FONT_16X26:ARRAY[0..255,0..51]OF BYTE :=[
16#00,16#00,16#00,16#00,16#00,16#00,16#00,16#00,16#00,16#00,16#00,16#00,16#00,16#00,16#00,16#00,16#00,16#00,16#00,16#00,16#00,16#00,16#00,16#00,16#00,16#00,16#00,16#00,16#00,16#00,16#00,16#00,16#00,16#00,16#00,16#00,16#00,16#00,16#00,16#00,16#00,16#00,16#00,16#00,16#00,16#00,16#00,16#00,16#00,16#00,16#00,16#00,	// 16#00
16#00,16#00,16#00,16#00,16#00,16#00,16#00,16#00,16#00,16#00,16#00,16#00,16#00,16#00,16#E0,16#07,16#30,16#0C,16#08,16#10,16#64,16#26,16#66,16#66,16#02,16#40,16#02,16#40,16#12,16#48,16#12,16#48,16#36,16#6C,16#24,16#24,16#C8,16#13,16#30,16#0C,16#E0,16#07,16#00,16#00,16#00,16#00,16#00,16#00,16#00,16#00,16#00,16#00,	// 16#01
16#00,16#00,16#00,16#00,16#00,16#00,16#00,16#00,16#00,16#00,16#00,16#00,16#00,16#00,16#E0,16#07,16#F0,16#0F,16#F8,16#1F,16#FC,16#3F,16#9E,16#79,16#9E,16#79,16#FE,16#7F,16#FE,16#7F,16#EE,16#77,16#EE,16#77,16#DC,16#3B,16#38,16#1C,16#F0,16#0F,16#E0,16#07,16#00,16#00,16#00,16#00,16#00,16#00,16#00,16#00,16#00,16#00,	// 16#02
16#00,16#00,16#00,16#00,16#3C,16#3C,16#7E,16#7E,16#FE,16#7F,16#FF,16#FF,16#FF,16#FF,16#FF,16#FF,16#FF,16#FF,16#FF,16#FF,16#FF,16#FF,16#FE,16#7F,16#FE,16#7F,16#FC,16#3F,16#FC,16#3F,16#F8,16#1F,16#F0,16#0F,16#F0,16#0F,16#E0,16#07,16#C0,16#03,16#80,16#01,16#00,16#00,16#00,16#00,16#00,16#00,16#00,16#00,16#00,16#00,	// 16#03
16#00,16#00,16#00,16#00,16#00,16#01,16#80,16#01,16#80,16#03,16#C0,16#07,16#E0,16#07,16#F0,16#0F,16#F8,16#1F,16#FC,16#3F,16#FE,16#7F,16#FF,16#FF,16#FE,16#7F,16#FC,16#3F,16#F8,16#1F,16#F0,16#0F,16#E0,16#07,16#C0,16#07,16#80,16#03,16#80,16#01,16#00,16#01,16#00,16#00,16#00,16#00,16#00,16#00,16#00,16#00,16#00,16#00,	// 16#04
16#00,16#00,16#00,16#00,16#C0,16#03,16#E0,16#07,16#F0,16#0F,16#F0,16#0F,16#F0,16#0F,16#F0,16#0F,16#E0,16#07,16#FC,16#3F,16#FE,16#7F,16#FF,16#FF,16#FF,16#FF,16#FF,16#FF,16#FE,16#7F,16#9C,16#39,16#80,16#01,16#80,16#01,16#C0,16#03,16#C0,16#03,16#C0,16#03,16#00,16#00,16#00,16#00,16#00,16#00,16#00,16#00,16#00,16#00,	// 16#05
16#00,16#00,16#00,16#00,16#80,16#00,16#80,16#01,16#C0,16#01,16#E0,16#03,16#F0,16#07,16#F0,16#0F,16#F8,16#1F,16#FC,16#3F,16#FE,16#7F,16#FF,16#7F,16#FF,16#FF,16#FF,16#FF,16#FF,16#FF,16#FE,16#7F,16#9C,16#39,16#80,16#01,16#80,16#01,16#C0,16#03,16#C0,16#03,16#00,16#00,16#00,16#00,16#00,16#00,16#00,16#00,16#00,16#00,	// 16#06
16#00,16#00,16#00,16#00,16#00,16#00,16#00,16#00,16#00,16#00,16#00,16#00,16#00,16#00,16#00,16#00,16#00,16#00,16#00,16#00,16#00,16#00,16#00,16#00,16#00,16#00,16#00,16#00,16#00,16#00,16#00,16#00,16#00,16#00,16#00,16#00,16#00,16#00,16#00,16#00,16#00,16#00,16#00,16#00,16#00,16#00,16#00,16#00,16#00,16#00,16#00,16#00,	// 16#07
16#00,16#00,16#00,16#00,16#00,16#00,16#00,16#00,16#00,16#00,16#00,16#00,16#00,16#00,16#00,16#00,16#00,16#00,16#00,16#00,16#00,16#00,16#00,16#00,16#00,16#00,16#00,16#00,16#00,16#00,16#00,16#00,16#00,16#00,16#00,16#00,16#00,16#00,16#00,16#00,16#00,16#00,16#00,16#00,16#00,16#00,16#00,16#00,16#00,16#00,16#00,16#00,	// 16#08
16#00,16#00,16#00,16#00,16#00,16#00,16#00,16#00,16#00,16#00,16#00,16#00,16#00,16#00,16#00,16#00,16#00,16#00,16#00,16#00,16#00,16#00,16#00,16#00,16#00,16#00,16#00,16#00,16#00,16#00,16#00,16#00,16#00,16#00,16#00,16#00,16#00,16#00,16#00,16#00,16#00,16#00,16#00,16#00,16#00,16#00,16#00,16#00,16#00,16#00,16#00,16#00,	// 16#09
16#00,16#00,16#00,16#00,16#00,16#00,16#00,16#00,16#00,16#00,16#00,16#00,16#00,16#00,16#00,16#00,16#00,16#00,16#00,16#00,16#00,16#00,16#00,16#00,16#00,16#00,16#00,16#00,16#00,16#00,16#00,16#00,16#00,16#00,16#00,16#00,16#00,16#00,16#00,16#00,16#00,16#00,16#00,16#00,16#00,16#00,16#00,16#00,16#00,16#00,16#00,16#00,	// 16#0A
16#00,16#00,16#00,16#00,16#0C,16#00,16#FE,16#00,16#FE,16#00,16#1E,16#00,16#33,16#00,16#73,16#00,16#E0,16#0F,16#E0,16#3F,16#70,16#70,16#30,16#60,16#18,16#C0,16#18,16#C0,16#18,16#C0,16#18,16#C0,16#18,16#C0,16#30,16#60,16#70,16#70,16#E0,16#3F,16#80,16#0F,16#00,16#00,16#00,16#00,16#00,16#00,16#00,16#00,16#00,16#00,	// 16#0B
16#00,16#00,16#00,16#00,16#E0,16#03,16#F8,16#0F,16#1C,16#1C,16#0C,16#18,16#06,16#30,16#06,16#30,16#06,16#30,16#06,16#30,16#06,16#38,16#0C,16#18,16#1C,16#1E,16#F8,16#0F,16#F0,16#03,16#C0,16#00,16#C0,16#00,16#F8,16#07,16#F8,16#07,16#C0,16#00,16#C0,16#00,16#00,16#00,16#00,16#00,16#00,16#00,16#00,16#00,16#00,16#00,	// 16#0C
16#00,16#00,16#00,16#00,16#00,16#00,16#00,16#00,16#00,16#00,16#00,16#00,16#00,16#00,16#00,16#00,16#00,16#00,16#00,16#00,16#00,16#00,16#00,16#00,16#00,16#00,16#00,16#00,16#00,16#00,16#00,16#00,16#00,16#00,16#00,16#00,16#00,16#00,16#00,16#00,16#00,16#00,16#00,16#00,16#00,16#00,16#00,16#00,16#00,16#00,16#00,16#00,	// 16#0D
16#00,16#00,16#00,16#00,16#02,16#00,16#0E,16#00,16#7E,16#00,16#FE,16#01,16#E2,16#07,16#82,16#07,16#02,16#04,16#02,16#04,16#02,16#04,16#02,16#04,16#02,16#04,16#02,16#04,16#02,16#04,16#02,16#04,16#1E,16#04,16#3E,16#04,16#7E,16#04,16#7C,16#04,16#38,16#3C,16#00,16#7C,16#00,16#FC,16#00,16#F8,16#00,16#70,16#00,16#00,	// 16#0E
16#00,16#00,16#00,16#00,16#00,16#00,16#00,16#00,16#00,16#00,16#80,16#01,16#88,16#11,16#DC,16#3B,16#F8,16#1F,16#30,16#0C,16#18,16#18,16#1E,16#78,16#1E,16#78,16#18,16#18,16#30,16#0C,16#F8,16#1F,16#DC,16#3B,16#88,16#11,16#80,16#01,16#00,16#00,16#00,16#00,16#00,16#00,16#00,16#00,16#00,16#00,16#00,16#00,16#00,16#00,	// 16#0F
16#00,16#00,16#00,16#00,16#00,16#00,16#00,16#00,16#00,16#00,16#00,16#00,16#00,16#40,16#00,16#70,16#00,16#7C,16#00,16#7F,16#80,16#7F,16#E0,16#7F,16#F8,16#7F,16#FE,16#7F,16#F8,16#7F,16#E0,16#7F,16#80,16#7F,16#00,16#7F,16#00,16#7C,16#00,16#70,16#00,16#40,16#00,16#00,16#00,16#00,16#00,16#00,16#00,16#00,16#00,16#00,	// 16#10
16#00,16#00,16#00,16#00,16#00,16#00,16#00,16#00,16#00,16#00,16#00,16#00,16#02,16#00,16#0E,16#00,16#3E,16#00,16#FE,16#00,16#FE,16#01,16#FE,16#07,16#FE,16#1F,16#FE,16#7F,16#FE,16#1F,16#FE,16#07,16#FE,16#01,16#FE,16#00,16#3E,16#00,16#0E,16#00,16#02,16#00,16#00,16#00,16#00,16#00,16#00,16#00,16#00,16#00,16#00,16#00,	// 16#11
16#00,16#00,16#00,16#00,16#80,16#01,16#80,16#01,16#C0,16#03,16#E0,16#07,16#B0,16#0D,16#80,16#01,16#80,16#01,16#80,16#01,16#80,16#01,16#80,16#01,16#80,16#01,16#80,16#01,16#80,16#01,16#80,16#01,16#80,16#01,16#80,16#01,16#80,16#01,16#80,16#01,16#B0,16#0D,16#E0,16#07,16#C0,16#03,16#80,16#01,16#80,16#01,16#00,16#00,	// 16#12
16#00,16#00,16#00,16#00,16#38,16#0E,16#38,16#0E,16#38,16#0E,16#38,16#0E,16#38,16#0E,16#38,16#0E,16#38,16#0E,16#38,16#0E,16#38,16#0E,16#38,16#0E,16#38,16#0E,16#38,16#0E,16#38,16#0E,16#38,16#0E,16#00,16#00,16#00,16#00,16#38,16#0E,16#38,16#0E,16#38,16#0E,16#00,16#00,16#00,16#00,16#00,16#00,16#00,16#00,16#00,16#00,	// 16#13
16#00,16#00,16#00,16#00,16#F8,16#1F,16#F8,16#3F,16#18,16#7F,16#18,16#7F,16#18,16#7F,16#18,16#7F,16#18,16#7F,16#18,16#3F,16#18,16#1F,16#18,16#0F,16#18,16#03,16#18,16#03,16#18,16#03,16#18,16#03,16#18,16#03,16#18,16#03,16#18,16#03,16#18,16#03,16#18,16#03,16#18,16#03,16#18,16#03,16#18,16#03,16#18,16#03,16#00,16#00,	// 16#14
16#00,16#00,16#00,16#00,16#F8,16#03,16#F8,16#0F,16#08,16#1E,16#00,16#1C,16#00,16#1C,16#00,16#1E,16#80,16#0F,16#E0,16#07,16#F0,16#0F,16#78,16#0C,16#3C,16#1C,16#1C,16#1C,16#1C,16#1E,16#98,16#0F,16#F0,16#07,16#F0,16#01,16#78,16#00,16#3C,16#00,16#1C,16#00,16#1C,16#00,16#3C,16#18,16#F8,16#1F,16#E0,16#07,16#00,16#00,	// 16#15
16#00,16#00,16#00,16#00,16#00,16#00,16#00,16#00,16#00,16#00,16#00,16#00,16#00,16#00,16#00,16#00,16#FE,16#7F,16#FE,16#7F,16#FE,16#7F,16#FE,16#7F,16#FE,16#7F,16#00,16#00,16#00,16#00,16#00,16#00,16#00,16#00,16#00,16#00,16#00,16#00,16#00,16#00,16#00,16#00,16#00,16#00,16#00,16#00,16#00,16#00,16#00,16#00,16#00,16#00,	// 16#16
16#00,16#00,16#80,16#01,16#80,16#01,16#C0,16#03,16#E0,16#07,16#B0,16#0D,16#80,16#01,16#80,16#01,16#80,16#01,16#80,16#01,16#80,16#01,16#80,16#01,16#80,16#01,16#80,16#01,16#80,16#01,16#80,16#01,16#80,16#01,16#80,16#01,16#B0,16#0D,16#E0,16#07,16#C0,16#03,16#80,16#01,16#80,16#01,16#00,16#00,16#F0,16#0F,16#F0,16#0F,	// 16#17
16#00,16#00,16#00,16#00,16#80,16#01,16#80,16#01,16#C0,16#03,16#E0,16#07,16#B0,16#0D,16#80,16#01,16#80,16#01,16#80,16#01,16#80,16#01,16#80,16#01,16#80,16#01,16#80,16#01,16#80,16#01,16#80,16#01,16#80,16#01,16#80,16#01,16#80,16#01,16#80,16#01,16#80,16#01,16#80,16#01,16#80,16#01,16#80,16#01,16#80,16#01,16#00,16#00,	// 16#18
16#00,16#00,16#00,16#00,16#80,16#01,16#80,16#01,16#80,16#01,16#80,16#01,16#80,16#01,16#80,16#01,16#80,16#01,16#80,16#01,16#80,16#01,16#80,16#01,16#80,16#01,16#80,16#01,16#80,16#01,16#80,16#01,16#80,16#01,16#80,16#01,16#80,16#01,16#80,16#01,16#B0,16#0D,16#E0,16#07,16#C0,16#03,16#80,16#01,16#80,16#01,16#00,16#00,	// 16#19
16#00,16#00,16#00,16#00,16#00,16#00,16#00,16#00,16#00,16#00,16#00,16#00,16#00,16#00,16#00,16#00,16#00,16#00,16#20,16#00,16#30,16#00,16#18,16#00,16#FE,16#7F,16#FE,16#7F,16#18,16#00,16#30,16#00,16#20,16#00,16#00,16#00,16#00,16#00,16#00,16#00,16#00,16#00,16#00,16#00,16#00,16#00,16#00,16#00,16#00,16#00,16#00,16#00,	// 16#1A
16#00,16#00,16#00,16#00,16#00,16#00,16#00,16#00,16#00,16#00,16#00,16#00,16#00,16#00,16#00,16#00,16#00,16#00,16#00,16#04,16#00,16#0C,16#00,16#18,16#FE,16#7F,16#FE,16#7F,16#00,16#18,16#00,16#0C,16#00,16#04,16#00,16#00,16#00,16#00,16#00,16#00,16#00,16#00,16#00,16#00,16#00,16#00,16#00,16#00,16#00,16#00,16#00,16#00,	// 16#1B
16#00,16#00,16#00,16#00,16#00,16#00,16#00,16#00,16#00,16#00,16#00,16#00,16#00,16#00,16#00,16#60,16#00,16#60,16#00,16#60,16#00,16#60,16#00,16#60,16#00,16#60,16#00,16#60,16#00,16#60,16#00,16#60,16#00,16#60,16#00,16#60,16#00,16#60,16#FE,16#7F,16#FE,16#7F,16#00,16#00,16#00,16#00,16#00,16#00,16#00,16#00,16#00,16#00,	// 16#1C
16#00,16#00,16#00,16#00,16#00,16#00,16#00,16#00,16#00,16#00,16#00,16#00,16#00,16#00,16#00,16#00,16#00,16#00,16#20,16#04,16#30,16#0C,16#18,16#18,16#FE,16#7F,16#FE,16#7F,16#18,16#18,16#30,16#0C,16#20,16#04,16#00,16#00,16#00,16#00,16#00,16#00,16#00,16#00,16#00,16#00,16#00,16#00,16#00,16#00,16#00,16#00,16#00,16#00,	// 16#1D
16#00,16#00,16#00,16#00,16#00,16#00,16#00,16#00,16#00,16#00,16#00,16#00,16#80,16#00,16#80,16#00,16#C0,16#01,16#C0,16#01,16#C0,16#03,16#E0,16#03,16#E0,16#07,16#F0,16#07,16#F0,16#0F,16#F8,16#0F,16#F8,16#1F,16#F8,16#1F,16#FC,16#3F,16#FC,16#3F,16#FE,16#7F,16#00,16#00,16#00,16#00,16#00,16#00,16#00,16#00,16#00,16#00,	// 16#1E
16#00,16#00,16#00,16#00,16#00,16#00,16#00,16#00,16#00,16#00,16#00,16#00,16#FE,16#7F,16#FC,16#3F,16#FC,16#3F,16#F8,16#1F,16#F8,16#1F,16#F8,16#0F,16#F0,16#0F,16#F0,16#07,16#E0,16#07,16#E0,16#03,16#C0,16#03,16#C0,16#01,16#C0,16#01,16#80,16#00,16#80,16#00,16#00,16#00,16#00,16#00,16#00,16#00,16#00,16#00,16#00,16#00,	// 16#1F
16#00,16#00,16#00,16#00,16#00,16#00,16#00,16#00,16#00,16#00,16#00,16#00,16#00,16#00,16#00,16#00,16#00,16#00,16#00,16#00,16#00,16#00,16#00,16#00,16#00,16#00,16#00,16#00,16#00,16#00,16#00,16#00,16#00,16#00,16#00,16#00,16#00,16#00,16#00,16#00,16#00,16#00,16#00,16#00,16#00,16#00,16#00,16#00,16#00,16#00,16#00,16#00,	// 16#20
16#00,16#00,16#00,16#00,16#C0,16#01,16#C0,16#01,16#C0,16#01,16#C0,16#01,16#C0,16#01,16#C0,16#01,16#C0,16#01,16#C0,16#01,16#C0,16#01,16#C0,16#01,16#C0,16#01,16#C0,16#01,16#C0,16#01,16#C0,16#01,16#00,16#00,16#00,16#00,16#C0,16#01,16#C0,16#01,16#C0,16#01,16#00,16#00,16#00,16#00,16#00,16#00,16#00,16#00,16#00,16#00,	// 16#21
16#00,16#00,16#70,16#1C,16#70,16#1C,16#70,16#1C,16#70,16#1C,16#70,16#1C,16#20,16#08,16#20,16#08,16#00,16#00,16#00,16#00,16#00,16#00,16#00,16#00,16#00,16#00,16#00,16#00,16#00,16#00,16#00,16#00,16#00,16#00,16#00,16#00,16#00,16#00,16#00,16#00,16#00,16#00,16#00,16#00,16#00,16#00,16#00,16#00,16#00,16#00,16#00,16#00,	// 16#22
16#00,16#00,16#00,16#00,16#8C,16#01,16#8C,16#01,16#18,16#03,16#18,16#03,16#18,16#03,16#18,16#03,16#FE,16#3F,16#FE,16#3F,16#30,16#06,16#60,16#06,16#60,16#0C,16#FC,16#7F,16#FC,16#7F,16#C0,16#18,16#C0,16#18,16#C0,16#18,16#C0,16#18,16#80,16#31,16#80,16#31,16#00,16#00,16#00,16#00,16#00,16#00,16#00,16#00,16#00,16#00,	// 16#23
16#C0,16#00,16#C0,16#00,16#F8,16#03,16#FC,16#0F,16#C4,16#0E,16#C0,16#1C,16#C0,16#1C,16#C0,16#1C,16#C0,16#1E,16#C0,16#0F,16#C0,16#07,16#E0,16#01,16#F8,16#00,16#F8,16#00,16#DC,16#00,16#DC,16#00,16#DC,16#00,16#DC,16#00,16#D8,16#18,16#F8,16#1F,16#F0,16#07,16#C0,16#00,16#C0,16#00,16#00,16#00,16#00,16#00,16#00,16#00,	// 16#24
16#00,16#00,16#00,16#00,16#03,16#3C,16#06,16#66,16#0C,16#C3,16#18,16#C3,16#18,16#C3,16#30,16#C3,16#60,16#C3,16#C0,16#66,16#C0,16#3C,16#80,16#01,16#3C,16#03,16#66,16#03,16#C3,16#06,16#C3,16#0C,16#C3,16#18,16#C3,16#18,16#C3,16#30,16#66,16#60,16#3C,16#C0,16#00,16#00,16#00,16#00,16#00,16#00,16#00,16#00,16#00,16#00,	// 16#25
16#00,16#00,16#00,16#00,16#C0,16#07,16#E0,16#0F,16#70,16#1C,16#70,16#1C,16#70,16#1C,16#60,16#1C,16#E0,16#0E,16#80,16#0F,16#00,16#1F,16#07,16#3F,16#87,16#73,16#C7,16#E3,16#C6,16#E1,16#E6,16#E0,16#7E,16#E0,16#7C,16#F0,16#3C,16#78,16#FE,16#3F,16#CF,16#0F,16#00,16#00,16#00,16#00,16#00,16#00,16#00,16#00,16#00,16#00,	// 16#26
16#00,16#00,16#80,16#03,16#80,16#03,16#80,16#03,16#80,16#03,16#80,16#03,16#00,16#01,16#00,16#01,16#00,16#00,16#00,16#00,16#00,16#00,16#00,16#00,16#00,16#00,16#00,16#00,16#00,16#00,16#00,16#00,16#00,16#00,16#00,16#00,16#00,16#00,16#00,16#00,16#00,16#00,16#00,16#00,16#00,16#00,16#00,16#00,16#00,16#00,16#00,16#00,	// 16#27
16#00,16#00,16#18,16#00,16#78,16#00,16#F0,16#00,16#C0,16#01,16#80,16#03,16#00,16#07,16#00,16#07,16#00,16#07,16#00,16#0E,16#00,16#0E,16#00,16#0E,16#00,16#0E,16#00,16#0E,16#00,16#0E,16#00,16#0E,16#00,16#0E,16#00,16#07,16#00,16#07,16#00,16#07,16#80,16#03,16#C0,16#01,16#F0,16#00,16#78,16#00,16#18,16#00,16#00,16#00,	// 16#28
16#00,16#00,16#00,16#30,16#00,16#3C,16#00,16#1E,16#00,16#07,16#80,16#03,16#C0,16#01,16#C0,16#01,16#C0,16#01,16#E0,16#00,16#E0,16#00,16#E0,16#00,16#E0,16#00,16#E0,16#00,16#E0,16#00,16#E0,16#00,16#E0,16#00,16#C0,16#01,16#C0,16#01,16#C0,16#01,16#80,16#03,16#00,16#07,16#00,16#1E,16#00,16#3C,16#00,16#30,16#00,16#00,	// 16#29
16#00,16#00,16#00,16#00,16#C0,16#01,16#C0,16#01,16#C0,16#01,16#D8,16#19,16#7C,16#3E,16#30,16#0C,16#40,16#02,16#E0,16#07,16#70,16#0E,16#38,16#1C,16#20,16#04,16#00,16#00,16#00,16#00,16#00,16#00,16#00,16#00,16#00,16#00,16#00,16#00,16#00,16#00,16#00,16#00,16#00,16#00,16#00,16#00,16#00,16#00,16#00,16#00,16#00,16#00,	// 16#2A
16#00,16#00,16#00,16#00,16#00,16#00,16#00,16#00,16#00,16#00,16#00,16#00,16#00,16#00,16#80,16#01,16#80,16#01,16#80,16#01,16#80,16#01,16#80,16#01,16#80,16#01,16#FE,16#7F,16#FE,16#7F,16#80,16#01,16#80,16#01,16#80,16#01,16#80,16#01,16#80,16#01,16#80,16#01,16#00,16#00,16#00,16#00,16#00,16#00,16#00,16#00,16#00,16#00,	// 16#2B
16#00,16#00,16#00,16#00,16#00,16#00,16#00,16#00,16#00,16#00,16#00,16#00,16#00,16#00,16#00,16#00,16#00,16#00,16#00,16#00,16#00,16#00,16#00,16#00,16#00,16#00,16#00,16#00,16#00,16#00,16#00,16#00,16#00,16#00,16#C0,16#03,16#C0,16#03,16#C0,16#03,16#C0,16#03,16#C0,16#00,16#C0,16#01,16#80,16#01,16#00,16#03,16#00,16#00,	// 16#2C
16#00,16#00,16#00,16#00,16#00,16#00,16#00,16#00,16#00,16#00,16#00,16#00,16#00,16#00,16#00,16#00,16#00,16#00,16#00,16#00,16#00,16#00,16#00,16#00,16#F8,16#1F,16#F8,16#1F,16#00,16#00,16#00,16#00,16#00,16#00,16#00,16#00,16#00,16#00,16#00,16#00,16#00,16#00,16#00,16#00,16#00,16#00,16#00,16#00,16#00,16#00,16#00,16#00,	// 16#2D
16#00,16#00,16#00,16#00,16#00,16#00,16#00,16#00,16#00,16#00,16#00,16#00,16#00,16#00,16#00,16#00,16#00,16#00,16#00,16#00,16#00,16#00,16#00,16#00,16#00,16#00,16#00,16#00,16#00,16#00,16#00,16#00,16#00,16#00,16#C0,16#03,16#C0,16#03,16#C0,16#03,16#C0,16#03,16#00,16#00,16#00,16#00,16#00,16#00,16#00,16#00,16#00,16#00,	// 16#2E
16#00,16#00,16#06,16#00,16#0C,16#00,16#0C,16#00,16#18,16#00,16#18,16#00,16#30,16#00,16#30,16#00,16#60,16#00,16#60,16#00,16#C0,16#00,16#C0,16#00,16#80,16#01,16#80,16#01,16#00,16#03,16#00,16#03,16#00,16#06,16#00,16#06,16#00,16#0C,16#00,16#0C,16#00,16#18,16#00,16#18,16#00,16#30,16#00,16#30,16#00,16#60,16#00,16#00,	// 16#2F
16#00,16#00,16#00,16#00,16#C0,16#07,16#E0,16#0F,16#70,16#1C,16#38,16#38,16#38,16#38,16#1C,16#70,16#1C,16#70,16#1C,16#70,16#1C,16#70,16#1C,16#70,16#1C,16#70,16#1C,16#70,16#1C,16#70,16#1C,16#70,16#38,16#38,16#38,16#38,16#70,16#1C,16#E0,16#0F,16#C0,16#07,16#00,16#00,16#00,16#00,16#00,16#00,16#00,16#00,16#00,16#00,	// 16#30
16#00,16#00,16#00,16#00,16#C0,16#00,16#C0,16#07,16#C0,16#3F,16#C0,16#31,16#C0,16#01,16#C0,16#01,16#C0,16#01,16#C0,16#01,16#C0,16#01,16#C0,16#01,16#C0,16#01,16#C0,16#01,16#C0,16#01,16#C0,16#01,16#C0,16#01,16#C0,16#01,16#C0,16#01,16#FE,16#3F,16#FE,16#3F,16#00,16#00,16#00,16#00,16#00,16#00,16#00,16#00,16#00,16#00,	// 16#31
16#00,16#00,16#00,16#00,16#C0,16#0F,16#E0,16#3F,16#70,16#30,16#38,16#00,16#38,16#00,16#38,16#00,16#38,16#00,16#70,16#00,16#70,16#00,16#E0,16#00,16#C0,16#01,16#80,16#03,16#00,16#07,16#00,16#0E,16#00,16#0C,16#00,16#1C,16#00,16#38,16#F8,16#3F,16#F8,16#3F,16#00,16#00,16#00,16#00,16#00,16#00,16#00,16#00,16#00,16#00,	// 16#32
16#00,16#00,16#00,16#00,16#C0,16#0F,16#F0,16#1F,16#78,16#10,16#38,16#00,16#38,16#00,16#38,16#00,16#30,16#00,16#60,16#00,16#C0,16#07,16#E0,16#07,16#F0,16#00,16#78,16#00,16#38,16#00,16#38,16#00,16#38,16#00,16#78,16#00,16#F0,16#10,16#E0,16#1F,16#C0,16#1F,16#00,16#00,16#00,16#00,16#00,16#00,16#00,16#00,16#00,16#00,	// 16#33
16#00,16#00,16#00,16#00,16#70,16#00,16#F0,16#00,16#F0,16#01,16#F0,16#01,16#70,16#03,16#70,16#07,16#70,16#06,16#70,16#0C,16#70,16#18,16#70,16#18,16#70,16#30,16#70,16#60,16#FE,16#7F,16#FE,16#7F,16#70,16#00,16#70,16#00,16#70,16#00,16#70,16#00,16#70,16#00,16#00,16#00,16#00,16#00,16#00,16#00,16#00,16#00,16#00,16#00,	// 16#34
16#00,16#00,16#00,16#00,16#FC,16#0F,16#FC,16#0F,16#FC,16#0F,16#00,16#0C,16#00,16#0C,16#00,16#0C,16#00,16#0C,16#00,16#0C,16#C0,16#0F,16#F0,16#0F,16#78,16#00,16#3C,16#00,16#1C,16#00,16#1C,16#00,16#1C,16#00,16#3C,16#00,16#78,16#08,16#F0,16#0F,16#C0,16#0F,16#00,16#00,16#00,16#00,16#00,16#00,16#00,16#00,16#00,16#00,	// 16#35
16#00,16#00,16#00,16#00,16#F8,16#01,16#FC,16#07,16#04,16#0F,16#00,16#0E,16#00,16#1C,16#00,16#1C,16#00,16#38,16#F0,16#39,16#F8,16#3B,16#3C,16#3E,16#1E,16#3C,16#0E,16#38,16#0E,16#38,16#0E,16#38,16#0E,16#1C,16#1C,16#1C,16#1C,16#0E,16#F8,16#0F,16#E0,16#03,16#00,16#00,16#00,16#00,16#00,16#00,16#00,16#00,16#00,16#00,	// 16#36
16#00,16#00,16#00,16#00,16#FC,16#1F,16#FC,16#1F,16#FC,16#1F,16#18,16#00,16#18,16#00,16#30,16#00,16#30,16#00,16#60,16#00,16#40,16#00,16#C0,16#00,16#80,16#01,16#80,16#01,16#00,16#03,16#00,16#03,16#00,16#06,16#00,16#06,16#00,16#0E,16#00,16#0C,16#00,16#0C,16#00,16#00,16#00,16#00,16#00,16#00,16#00,16#00,16#00,16#00,	// 16#37
16#00,16#00,16#00,16#00,16#E0,16#03,16#F0,16#0F,16#78,16#1E,16#38,16#1C,16#38,16#1C,16#38,16#1C,16#30,16#1E,16#F0,16#0F,16#C0,16#07,16#F0,16#0F,16#F8,16#1C,16#78,16#18,16#3C,16#38,16#1C,16#38,16#1C,16#38,16#1C,16#38,16#38,16#1C,16#F0,16#0F,16#E0,16#07,16#00,16#00,16#00,16#00,16#00,16#00,16#00,16#00,16#00,16#00,	// 16#38
16#00,16#00,16#00,16#00,16#E0,16#03,16#F8,16#0F,16#38,16#1C,16#1C,16#1C,16#1C,16#38,16#0E,16#38,16#0E,16#38,16#0E,16#38,16#1E,16#3C,16#3E,16#1E,16#EE,16#0F,16#CE,16#07,16#0E,16#00,16#1C,16#00,16#1C,16#00,16#38,16#00,16#78,16#10,16#F0,16#1F,16#C0,16#0F,16#00,16#00,16#00,16#00,16#00,16#00,16#00,16#00,16#00,16#00,	// 16#39
16#00,16#00,16#00,16#00,16#00,16#00,16#00,16#00,16#00,16#00,16#00,16#00,16#00,16#00,16#C0,16#03,16#C0,16#03,16#C0,16#03,16#C0,16#03,16#00,16#00,16#00,16#00,16#00,16#00,16#00,16#00,16#00,16#00,16#00,16#00,16#C0,16#03,16#C0,16#03,16#C0,16#03,16#C0,16#03,16#00,16#00,16#00,16#00,16#00,16#00,16#00,16#00,16#00,16#00,	// 16#3A
16#00,16#00,16#00,16#00,16#00,16#00,16#00,16#00,16#00,16#00,16#00,16#00,16#00,16#00,16#C0,16#03,16#C0,16#03,16#C0,16#03,16#C0,16#03,16#00,16#00,16#00,16#00,16#00,16#00,16#00,16#00,16#00,16#00,16#00,16#00,16#C0,16#03,16#C0,16#03,16#C0,16#03,16#C0,16#03,16#C0,16#00,16#C0,16#01,16#80,16#01,16#00,16#03,16#00,16#00,	// 16#3B
16#00,16#00,16#00,16#00,16#00,16#00,16#00,16#00,16#00,16#00,16#00,16#00,16#00,16#00,16#02,16#00,16#0E,16#00,16#3C,16#00,16#F0,16#00,16#C0,16#03,16#00,16#0F,16#00,16#3C,16#00,16#3C,16#00,16#0F,16#C0,16#03,16#F0,16#00,16#3C,16#00,16#0E,16#00,16#02,16#00,16#00,16#00,16#00,16#00,16#00,16#00,16#00,16#00,16#00,16#00,	// 16#3C
16#00,16#00,16#00,16#00,16#00,16#00,16#00,16#00,16#00,16#00,16#00,16#00,16#00,16#00,16#00,16#00,16#00,16#00,16#00,16#00,16#FE,16#7F,16#FE,16#7F,16#00,16#00,16#00,16#00,16#00,16#00,16#FE,16#7F,16#FE,16#7F,16#00,16#00,16#00,16#00,16#00,16#00,16#00,16#00,16#00,16#00,16#00,16#00,16#00,16#00,16#00,16#00,16#00,16#00,	// 16#3D
16#00,16#00,16#00,16#00,16#00,16#00,16#00,16#00,16#00,16#00,16#00,16#00,16#00,16#00,16#00,16#40,16#00,16#70,16#00,16#3C,16#00,16#0F,16#C0,16#03,16#F0,16#00,16#3C,16#00,16#3C,16#00,16#F0,16#00,16#C0,16#03,16#00,16#0F,16#00,16#3C,16#00,16#70,16#00,16#40,16#00,16#00,16#00,16#00,16#00,16#00,16#00,16#00,16#00,16#00,	// 16#3E
16#00,16#00,16#00,16#00,16#E0,16#1F,16#F8,16#3F,16#3C,16#30,16#1C,16#30,16#1C,16#00,16#1C,16#00,16#38,16#00,16#78,16#00,16#F0,16#00,16#E0,16#01,16#C0,16#01,16#80,16#03,16#80,16#03,16#80,16#03,16#00,16#00,16#00,16#00,16#80,16#03,16#80,16#03,16#80,16#03,16#00,16#00,16#00,16#00,16#00,16#00,16#00,16#00,16#00,16#00,	// 16#3F
16#00,16#00,16#00,16#00,16#F0,16#03,16#F8,16#07,16#1C,16#0E,16#0C,16#18,16#7C,16#38,16#8C,16#30,16#8C,16#71,16#0C,16#63,16#0C,16#63,16#1C,16#63,16#1C,16#63,16#3C,16#63,16#2C,16#63,16#EF,16#71,16#CF,16#31,16#00,16#38,16#10,16#1C,16#F0,16#0F,16#E0,16#03,16#00,16#00,16#00,16#00,16#00,16#00,16#00,16#00,16#00,16#00,	// 16#40
16#00,16#00,16#00,16#00,16#00,16#00,16#00,16#00,16#00,16#00,16#80,16#03,16#C0,16#03,16#C0,16#07,16#E0,16#06,16#E0,16#06,16#60,16#0E,16#70,16#0C,16#70,16#1C,16#38,16#1C,16#38,16#18,16#FC,16#3F,16#FC,16#3F,16#1C,16#70,16#0E,16#70,16#0E,16#70,16#07,16#E0,16#00,16#00,16#00,16#00,16#00,16#00,16#00,16#00,16#00,16#00,	// 16#41
16#00,16#00,16#00,16#00,16#00,16#00,16#00,16#00,16#00,16#00,16#E0,16#3F,16#F0,16#3F,16#78,16#38,16#38,16#38,16#38,16#38,16#70,16#38,16#E0,16#3F,16#E0,16#3F,16#78,16#38,16#3C,16#38,16#1C,16#38,16#1C,16#38,16#1C,16#38,16#3C,16#38,16#F8,16#3F,16#E0,16#3F,16#00,16#00,16#00,16#00,16#00,16#00,16#00,16#00,16#00,16#00,	// 16#42
16#00,16#00,16#00,16#00,16#00,16#00,16#00,16#00,16#00,16#00,16#F8,16#03,16#FC,16#0F,16#0C,16#1E,16#00,16#3C,16#00,16#38,16#00,16#70,16#00,16#70,16#00,16#70,16#00,16#70,16#00,16#70,16#00,16#70,16#00,16#38,16#00,16#3C,16#04,16#1E,16#FC,16#0F,16#F8,16#03,16#00,16#00,16#00,16#00,16#00,16#00,16#00,16#00,16#00,16#00,	// 16#43
16#00,16#00,16#00,16#00,16#00,16#00,16#00,16#00,16#00,16#00,16#E0,16#3F,16#F0,16#3F,16#3C,16#38,16#1C,16#38,16#1E,16#38,16#0E,16#38,16#0E,16#38,16#0E,16#38,16#0E,16#38,16#0E,16#38,16#0E,16#38,16#1C,16#38,16#1C,16#38,16#78,16#38,16#F0,16#3F,16#C0,16#3F,16#00,16#00,16#00,16#00,16#00,16#00,16#00,16#00,16#00,16#00,	// 16#44
16#00,16#00,16#00,16#00,16#00,16#00,16#00,16#00,16#00,16#00,16#FC,16#1F,16#FC,16#1F,16#00,16#1C,16#00,16#1C,16#00,16#1C,16#00,16#1C,16#00,16#1C,16#F8,16#1F,16#F8,16#1F,16#00,16#1C,16#00,16#1C,16#00,16#1C,16#00,16#1C,16#00,16#1C,16#FE,16#1F,16#FE,16#1F,16#00,16#00,16#00,16#00,16#00,16#00,16#00,16#00,16#00,16#00,	// 16#45
16#00,16#00,16#00,16#00,16#00,16#00,16#00,16#00,16#00,16#00,16#FE,16#1F,16#FE,16#1F,16#00,16#1C,16#00,16#1C,16#00,16#1C,16#00,16#1C,16#00,16#1C,16#FC,16#1F,16#FC,16#1F,16#00,16#1C,16#00,16#1C,16#00,16#1C,16#00,16#1C,16#00,16#1C,16#00,16#1C,16#00,16#1C,16#00,16#00,16#00,16#00,16#00,16#00,16#00,16#00,16#00,16#00,	// 16#46
16#00,16#00,16#00,16#00,16#00,16#00,16#00,16#00,16#00,16#00,16#F8,16#03,16#FC,16#0F,16#0C,16#1E,16#00,16#3C,16#00,16#38,16#00,16#70,16#00,16#70,16#00,16#70,16#FC,16#70,16#FC,16#70,16#1C,16#70,16#1C,16#38,16#1C,16#3C,16#1C,16#1E,16#FC,16#0F,16#F8,16#03,16#00,16#00,16#00,16#00,16#00,16#00,16#00,16#00,16#00,16#00,	// 16#47
16#00,16#00,16#00,16#00,16#00,16#00,16#00,16#00,16#00,16#00,16#1C,16#38,16#1C,16#38,16#1C,16#38,16#1C,16#38,16#1C,16#38,16#1C,16#38,16#1C,16#38,16#FC,16#3F,16#FC,16#3F,16#1C,16#38,16#1C,16#38,16#1C,16#38,16#1C,16#38,16#1C,16#38,16#1C,16#38,16#1C,16#38,16#00,16#00,16#00,16#00,16#00,16#00,16#00,16#00,16#00,16#00,	// 16#48
16#00,16#00,16#00,16#00,16#00,16#00,16#00,16#00,16#00,16#00,16#F8,16#3F,16#F8,16#3F,16#80,16#03,16#80,16#03,16#80,16#03,16#80,16#03,16#80,16#03,16#80,16#03,16#80,16#03,16#80,16#03,16#80,16#03,16#80,16#03,16#80,16#03,16#80,16#03,16#F8,16#3F,16#F8,16#3F,16#00,16#00,16#00,16#00,16#00,16#00,16#00,16#00,16#00,16#00,	// 16#49
16#00,16#00,16#00,16#00,16#00,16#00,16#00,16#00,16#00,16#00,16#F0,16#1F,16#F0,16#1F,16#70,16#00,16#70,16#00,16#70,16#00,16#70,16#00,16#70,16#00,16#70,16#00,16#70,16#00,16#70,16#00,16#70,16#00,16#70,16#00,16#70,16#00,16#E0,16#20,16#C0,16#3F,16#80,16#3F,16#00,16#00,16#00,16#00,16#00,16#00,16#00,16#00,16#00,16#00,	// 16#4A
16#00,16#00,16#00,16#00,16#00,16#00,16#00,16#00,16#00,16#00,16#1E,16#38,16#3C,16#38,16#78,16#38,16#F0,16#38,16#E0,16#38,16#C0,16#39,16#80,16#3B,16#00,16#3F,16#80,16#3B,16#C0,16#3B,16#E0,16#39,16#F0,16#38,16#78,16#38,16#3C,16#38,16#1E,16#38,16#1F,16#38,16#00,16#00,16#00,16#00,16#00,16#00,16#00,16#00,16#00,16#00,	// 16#4B
16#00,16#00,16#00,16#00,16#00,16#00,16#00,16#00,16#00,16#00,16#00,16#1C,16#00,16#1C,16#00,16#1C,16#00,16#1C,16#00,16#1C,16#00,16#1C,16#00,16#1C,16#00,16#1C,16#00,16#1C,16#00,16#1C,16#00,16#1C,16#00,16#1C,16#00,16#1C,16#00,16#1C,16#FC,16#1F,16#FC,16#1F,16#00,16#00,16#00,16#00,16#00,16#00,16#00,16#00,16#00,16#00,	// 16#4C
16#00,16#00,16#00,16#00,16#00,16#00,16#00,16#00,16#00,16#00,16#1C,16#70,16#3C,16#78,16#3C,16#78,16#3C,16#78,16#6C,16#6C,16#6C,16#6C,16#6C,16#6C,16#4C,16#66,16#CC,16#66,16#CC,16#66,16#8C,16#63,16#8C,16#63,16#8C,16#63,16#0C,16#60,16#0C,16#60,16#0C,16#60,16#00,16#00,16#00,16#00,16#00,16#00,16#00,16#00,16#00,16#00,	// 16#4D
16#00,16#00,16#00,16#00,16#00,16#00,16#00,16#00,16#00,16#00,16#0C,16#38,16#0C,16#38,16#0C,16#3C,16#0C,16#3E,16#0C,16#3E,16#0C,16#3F,16#8C,16#37,16#8C,16#33,16#CC,16#33,16#EC,16#31,16#FC,16#30,16#7C,16#30,16#7C,16#30,16#3C,16#30,16#1C,16#30,16#1C,16#30,16#00,16#00,16#00,16#00,16#00,16#00,16#00,16#00,16#00,16#00,	// 16#4E
16#00,16#00,16#00,16#00,16#00,16#00,16#00,16#00,16#00,16#00,16#E0,16#07,16#F0,16#0F,16#38,16#1C,16#1C,16#38,16#1C,16#38,16#0E,16#70,16#0E,16#70,16#0E,16#70,16#0E,16#70,16#0E,16#70,16#0E,16#70,16#1C,16#38,16#1C,16#38,16#38,16#1C,16#F0,16#0F,16#E0,16#07,16#00,16#00,16#00,16#00,16#00,16#00,16#00,16#00,16#00,16#00,	// 16#4F
16#00,16#00,16#00,16#00,16#00,16#00,16#00,16#00,16#00,16#00,16#F8,16#1F,16#FC,16#1F,16#1E,16#1C,16#0E,16#1C,16#0E,16#1C,16#0E,16#1C,16#1E,16#1C,16#3C,16#1C,16#F8,16#1F,16#E0,16#1F,16#00,16#1C,16#00,16#1C,16#00,16#1C,16#00,16#1C,16#00,16#1C,16#00,16#1C,16#00,16#00,16#00,16#00,16#00,16#00,16#00,16#00,16#00,16#00,	// 16#50
16#00,16#00,16#00,16#00,16#00,16#00,16#00,16#00,16#00,16#00,16#E0,16#07,16#F0,16#0F,16#38,16#1C,16#1C,16#38,16#1C,16#38,16#0E,16#70,16#0E,16#70,16#0E,16#70,16#0E,16#70,16#0E,16#70,16#0E,16#70,16#1C,16#38,16#1C,16#38,16#38,16#1C,16#F0,16#0F,16#E0,16#07,16#78,16#00,16#1E,16#00,16#0F,16#00,16#02,16#00,16#00,16#00,	// 16#51
16#00,16#00,16#00,16#00,16#00,16#00,16#00,16#00,16#00,16#00,16#E0,16#3F,16#F0,16#3F,16#78,16#38,16#38,16#38,16#38,16#38,16#38,16#38,16#70,16#38,16#E0,16#3F,16#C0,16#3F,16#E0,16#39,16#E0,16#38,16#F0,16#38,16#78,16#38,16#3C,16#38,16#1C,16#38,16#1E,16#38,16#00,16#00,16#00,16#00,16#00,16#00,16#00,16#00,16#00,16#00,	// 16#52
16#00,16#00,16#00,16#00,16#00,16#00,16#00,16#00,16#00,16#00,16#F0,16#07,16#F8,16#1F,16#18,16#3C,16#00,16#38,16#00,16#38,16#00,16#3C,16#00,16#1F,16#E0,16#0F,16#F8,16#03,16#7C,16#00,16#1C,16#00,16#1C,16#00,16#1C,16#00,16#38,16#30,16#F8,16#3F,16#E0,16#0F,16#00,16#00,16#00,16#00,16#00,16#00,16#00,16#00,16#00,16#00,	// 16#53
16#00,16#00,16#00,16#00,16#00,16#00,16#00,16#00,16#00,16#00,16#FE,16#FF,16#FE,16#FF,16#80,16#03,16#80,16#03,16#80,16#03,16#80,16#03,16#80,16#03,16#80,16#03,16#80,16#03,16#80,16#03,16#80,16#03,16#80,16#03,16#80,16#03,16#80,16#03,16#80,16#03,16#80,16#03,16#00,16#00,16#00,16#00,16#00,16#00,16#00,16#00,16#00,16#00,	// 16#54
16#00,16#00,16#00,16#00,16#00,16#00,16#00,16#00,16#00,16#00,16#0E,16#38,16#0E,16#38,16#0E,16#38,16#0E,16#38,16#0E,16#38,16#0E,16#38,16#0E,16#38,16#0E,16#38,16#0E,16#38,16#0E,16#38,16#0E,16#38,16#0E,16#38,16#1E,16#3C,16#1C,16#1C,16#F8,16#0F,16#F0,16#07,16#00,16#00,16#00,16#00,16#00,16#00,16#00,16#00,16#00,16#00,	// 16#55
16#00,16#00,16#00,16#00,16#00,16#00,16#00,16#00,16#00,16#00,16#07,16#E0,16#0E,16#70,16#0E,16#70,16#0E,16#38,16#1C,16#38,16#1C,16#3C,16#1C,16#1C,16#38,16#1C,16#38,16#0E,16#30,16#0E,16#70,16#07,16#70,16#07,16#E0,16#07,16#E0,16#03,16#E0,16#03,16#C0,16#01,16#00,16#00,16#00,16#00,16#00,16#00,16#00,16#00,16#00,16#00,	// 16#56
16#00,16#00,16#00,16#00,16#00,16#00,16#00,16#00,16#00,16#00,16#03,16#C0,16#03,16#C0,16#03,16#E0,16#86,16#61,16#C6,16#63,16#C6,16#63,16#C6,16#63,16#C6,16#63,16#6E,16#72,16#6C,16#36,16#6C,16#36,16#6C,16#36,16#7C,16#34,16#3C,16#3C,16#38,16#3C,16#38,16#3C,16#00,16#00,16#00,16#00,16#00,16#00,16#00,16#00,16#00,16#00,	// 16#57
16#00,16#00,16#00,16#00,16#00,16#00,16#00,16#00,16#00,16#00,16#07,16#78,16#0E,16#3C,16#1C,16#1E,16#38,16#1E,16#70,16#0F,16#E0,16#07,16#C0,16#03,16#C0,16#03,16#E0,16#03,16#E0,16#07,16#F0,16#06,16#78,16#0C,16#3C,16#18,16#1C,16#38,16#1E,16#70,16#0F,16#E0,16#00,16#00,16#00,16#00,16#00,16#00,16#00,16#00,16#00,16#00,	// 16#58
16#00,16#00,16#00,16#00,16#00,16#00,16#00,16#00,16#00,16#00,16#07,16#E0,16#0E,16#70,16#0C,16#38,16#18,16#38,16#38,16#1C,16#70,16#1E,16#E0,16#0E,16#C0,16#07,16#C0,16#07,16#80,16#03,16#80,16#03,16#80,16#03,16#80,16#03,16#80,16#03,16#80,16#03,16#80,16#03,16#00,16#00,16#00,16#00,16#00,16#00,16#00,16#00,16#00,16#00,	// 16#59
16#00,16#00,16#00,16#00,16#00,16#00,16#00,16#00,16#00,16#00,16#FC,16#3F,16#FC,16#3F,16#1C,16#00,16#38,16#00,16#70,16#00,16#E0,16#00,16#C0,16#01,16#80,16#01,16#00,16#03,16#00,16#07,16#00,16#0E,16#00,16#1C,16#00,16#38,16#00,16#70,16#FC,16#7F,16#FC,16#7F,16#00,16#00,16#00,16#00,16#00,16#00,16#00,16#00,16#00,16#00,	// 16#5A
16#00,16#00,16#FC,16#03,16#FC,16#03,16#80,16#03,16#80,16#03,16#80,16#03,16#80,16#03,16#80,16#03,16#80,16#03,16#80,16#03,16#80,16#03,16#80,16#03,16#80,16#03,16#80,16#03,16#80,16#03,16#80,16#03,16#80,16#03,16#80,16#03,16#80,16#03,16#80,16#03,16#80,16#03,16#80,16#03,16#80,16#03,16#FC,16#03,16#FC,16#03,16#00,16#00,	// 16#5B
16#00,16#00,16#00,16#60,16#00,16#30,16#00,16#30,16#00,16#18,16#00,16#18,16#00,16#0C,16#00,16#0C,16#00,16#06,16#00,16#06,16#00,16#03,16#00,16#03,16#80,16#01,16#80,16#01,16#C0,16#00,16#C0,16#00,16#60,16#00,16#60,16#00,16#30,16#00,16#30,16#00,16#18,16#00,16#18,16#00,16#0C,16#00,16#0C,16#00,16#06,16#00,16#00,16#00,	// 16#5C
16#00,16#00,16#C0,16#3F,16#C0,16#3F,16#C0,16#01,16#C0,16#01,16#C0,16#01,16#C0,16#01,16#C0,16#01,16#C0,16#01,16#C0,16#01,16#C0,16#01,16#C0,16#01,16#C0,16#01,16#C0,16#01,16#C0,16#01,16#C0,16#01,16#C0,16#01,16#C0,16#01,16#C0,16#01,16#C0,16#01,16#C0,16#01,16#C0,16#01,16#C0,16#01,16#C0,16#3F,16#C0,16#3F,16#00,16#00,	// 16#5D
16#00,16#00,16#00,16#00,16#80,16#00,16#80,16#00,16#C0,16#01,16#C0,16#01,16#C0,16#03,16#60,16#03,16#60,16#07,16#30,16#06,16#30,16#0C,16#18,16#0C,16#18,16#18,16#18,16#18,16#0C,16#30,16#0C,16#30,16#06,16#60,16#00,16#00,16#00,16#00,16#00,16#00,16#00,16#00,16#00,16#00,16#00,16#00,16#00,16#00,16#00,16#00,16#00,16#00,	// 16#5E
16#00,16#00,16#00,16#00,16#00,16#00,16#00,16#00,16#00,16#00,16#00,16#00,16#00,16#00,16#00,16#00,16#00,16#00,16#00,16#00,16#00,16#00,16#00,16#00,16#00,16#00,16#00,16#00,16#00,16#00,16#00,16#00,16#00,16#00,16#00,16#00,16#00,16#00,16#00,16#00,16#00,16#00,16#FF,16#FF,16#FF,16#FF,16#00,16#00,16#00,16#00,16#00,16#00,	// 16#5F
16#80,16#03,16#C0,16#01,16#E0,16#00,16#00,16#00,16#00,16#00,16#00,16#00,16#00,16#00,16#00,16#00,16#00,16#00,16#00,16#00,16#00,16#00,16#00,16#00,16#00,16#00,16#00,16#00,16#00,16#00,16#00,16#00,16#00,16#00,16#00,16#00,16#00,16#00,16#00,16#00,16#00,16#00,16#00,16#00,16#00,16#00,16#00,16#00,16#00,16#00,16#00,16#00,	// 16#60
16#00,16#00,16#00,16#00,16#00,16#00,16#00,16#00,16#00,16#00,16#00,16#00,16#00,16#00,16#E0,16#07,16#F0,16#1F,16#78,16#18,16#38,16#00,16#38,16#00,16#F8,16#07,16#F8,16#0F,16#38,16#1C,16#38,16#38,16#38,16#38,16#38,16#38,16#78,16#3C,16#DE,16#1F,16#1E,16#0F,16#00,16#00,16#00,16#00,16#00,16#00,16#00,16#00,16#00,16#00,	// 16#61
16#00,16#00,16#00,16#38,16#00,16#38,16#00,16#38,16#00,16#38,16#00,16#38,16#00,16#38,16#E0,16#39,16#F8,16#3B,16#38,16#3E,16#1C,16#3C,16#1C,16#38,16#1C,16#38,16#1C,16#38,16#1C,16#38,16#1C,16#38,16#1C,16#38,16#38,16#38,16#78,16#3C,16#F0,16#3F,16#E0,16#33,16#00,16#00,16#00,16#00,16#00,16#00,16#00,16#00,16#00,16#00,	// 16#62
16#00,16#00,16#00,16#00,16#00,16#00,16#00,16#00,16#00,16#00,16#00,16#00,16#00,16#00,16#F8,16#03,16#FC,16#0F,16#04,16#1E,16#00,16#1C,16#00,16#38,16#00,16#38,16#00,16#38,16#00,16#38,16#00,16#38,16#00,16#3C,16#00,16#1C,16#04,16#1F,16#FC,16#0F,16#F8,16#03,16#00,16#00,16#00,16#00,16#00,16#00,16#00,16#00,16#00,16#00,	// 16#63
16#00,16#00,16#0E,16#00,16#0E,16#00,16#0E,16#00,16#0E,16#00,16#0E,16#00,16#0E,16#00,16#CE,16#03,16#FE,16#0F,16#3E,16#1E,16#0E,16#1C,16#0E,16#38,16#0E,16#38,16#0E,16#38,16#0E,16#38,16#0E,16#38,16#0E,16#38,16#1E,16#3C,16#3E,16#1C,16#EE,16#0F,16#CE,16#07,16#00,16#00,16#00,16#00,16#00,16#00,16#00,16#00,16#00,16#00,	// 16#64
16#00,16#00,16#00,16#00,16#00,16#00,16#00,16#00,16#00,16#00,16#00,16#00,16#00,16#00,16#E0,16#03,16#F0,16#0F,16#38,16#1E,16#1C,16#1C,16#1C,16#38,16#1C,16#38,16#FC,16#3F,16#FC,16#3F,16#00,16#38,16#00,16#38,16#00,16#1C,16#04,16#1E,16#FC,16#0F,16#F8,16#03,16#00,16#00,16#00,16#00,16#00,16#00,16#00,16#00,16#00,16#00,	// 16#65
16#00,16#00,16#FF,16#00,16#FF,16#01,16#C0,16#03,16#80,16#03,16#80,16#03,16#80,16#03,16#FE,16#3F,16#FE,16#3F,16#80,16#03,16#80,16#03,16#80,16#03,16#80,16#03,16#80,16#03,16#80,16#03,16#80,16#03,16#80,16#03,16#80,16#03,16#80,16#03,16#80,16#03,16#80,16#03,16#00,16#00,16#00,16#00,16#00,16#00,16#00,16#00,16#00,16#00,	// 16#66
16#00,16#00,16#00,16#00,16#00,16#00,16#00,16#00,16#00,16#00,16#00,16#00,16#00,16#00,16#CE,16#03,16#FE,16#0F,16#3E,16#1E,16#0E,16#1C,16#0E,16#38,16#0E,16#38,16#0E,16#38,16#0E,16#38,16#0E,16#38,16#0E,16#38,16#1E,16#3C,16#3E,16#1C,16#EE,16#0F,16#CE,16#07,16#0E,16#00,16#1C,16#00,16#3C,16#18,16#F8,16#1F,16#E0,16#0F,	// 16#67
16#00,16#00,16#00,16#38,16#00,16#38,16#00,16#38,16#00,16#38,16#00,16#38,16#00,16#38,16#F0,16#38,16#F8,16#3B,16#3C,16#3E,16#1C,16#3C,16#1C,16#38,16#1C,16#38,16#1C,16#38,16#1C,16#38,16#1C,16#38,16#1C,16#38,16#1C,16#38,16#1C,16#38,16#1C,16#38,16#1C,16#38,16#00,16#00,16#00,16#00,16#00,16#00,16#00,16#00,16#00,16#00,	// 16#68
16#00,16#00,16#C0,16#01,16#C0,16#01,16#C0,16#01,16#00,16#00,16#00,16#00,16#00,16#00,16#C0,16#3F,16#C0,16#3F,16#C0,16#01,16#C0,16#01,16#C0,16#01,16#C0,16#01,16#C0,16#01,16#C0,16#01,16#C0,16#01,16#C0,16#01,16#C0,16#01,16#C0,16#01,16#C0,16#01,16#C0,16#01,16#00,16#00,16#00,16#00,16#00,16#00,16#00,16#00,16#00,16#00,	// 16#69
16#00,16#00,16#70,16#00,16#70,16#00,16#70,16#00,16#00,16#00,16#00,16#00,16#00,16#00,16#F0,16#1F,16#F0,16#1F,16#70,16#00,16#70,16#00,16#70,16#00,16#70,16#00,16#70,16#00,16#70,16#00,16#70,16#00,16#70,16#00,16#70,16#00,16#70,16#00,16#70,16#00,16#70,16#00,16#70,16#00,16#70,16#00,16#E0,16#20,16#E0,16#3F,16#80,16#1F,	// 16#6A
16#00,16#00,16#00,16#1C,16#00,16#1C,16#00,16#1C,16#00,16#1C,16#00,16#1C,16#00,16#1C,16#3C,16#1C,16#78,16#1C,16#70,16#1C,16#F0,16#1C,16#E0,16#1D,16#C0,16#1D,16#C0,16#1F,16#C0,16#1D,16#E0,16#1D,16#F0,16#1C,16#70,16#1C,16#78,16#1C,16#3C,16#1C,16#1E,16#1C,16#00,16#00,16#00,16#00,16#00,16#00,16#00,16#00,16#00,16#00,	// 16#6B
16#00,16#00,16#E0,16#1F,16#E0,16#1F,16#E0,16#00,16#E0,16#00,16#E0,16#00,16#E0,16#00,16#E0,16#00,16#E0,16#00,16#E0,16#00,16#E0,16#00,16#E0,16#00,16#E0,16#00,16#E0,16#00,16#E0,16#00,16#E0,16#00,16#E0,16#00,16#E0,16#00,16#E0,16#00,16#E0,16#00,16#E0,16#00,16#00,16#00,16#00,16#00,16#00,16#00,16#00,16#00,16#00,16#00,	// 16#6C
16#00,16#00,16#00,16#00,16#00,16#00,16#00,16#00,16#00,16#00,16#00,16#00,16#00,16#00,16#8C,16#73,16#9E,16#77,16#FE,16#7F,16#EE,16#79,16#CE,16#79,16#CE,16#71,16#CE,16#71,16#CE,16#71,16#CE,16#71,16#CE,16#71,16#CE,16#71,16#CE,16#71,16#CE,16#71,16#CE,16#71,16#00,16#00,16#00,16#00,16#00,16#00,16#00,16#00,16#00,16#00,	// 16#6D
16#00,16#00,16#00,16#00,16#00,16#00,16#00,16#00,16#00,16#00,16#00,16#00,16#00,16#00,16#F0,16#38,16#F8,16#3B,16#3C,16#3E,16#1C,16#3C,16#1C,16#38,16#1C,16#38,16#1C,16#38,16#1C,16#38,16#1C,16#38,16#1C,16#38,16#1C,16#38,16#1C,16#38,16#1C,16#38,16#1C,16#38,16#00,16#00,16#00,16#00,16#00,16#00,16#00,16#00,16#00,16#00,	// 16#6E
16#00,16#00,16#00,16#00,16#00,16#00,16#00,16#00,16#00,16#00,16#00,16#00,16#00,16#00,16#C0,16#07,16#F0,16#1F,16#78,16#3C,16#38,16#38,16#1C,16#70,16#1C,16#70,16#1C,16#70,16#1C,16#70,16#1C,16#70,16#1C,16#70,16#38,16#38,16#78,16#3C,16#F0,16#1F,16#C0,16#07,16#00,16#00,16#00,16#00,16#00,16#00,16#00,16#00,16#00,16#00,	// 16#6F
16#00,16#00,16#00,16#00,16#00,16#00,16#00,16#00,16#00,16#00,16#00,16#00,16#00,16#00,16#E0,16#39,16#F8,16#3B,16#38,16#3E,16#1C,16#3C,16#1C,16#38,16#1C,16#38,16#1C,16#38,16#1C,16#38,16#1C,16#38,16#1C,16#38,16#38,16#38,16#78,16#3C,16#F0,16#3F,16#E0,16#39,16#00,16#38,16#00,16#38,16#00,16#38,16#00,16#38,16#00,16#38,	// 16#70
16#00,16#00,16#00,16#00,16#00,16#00,16#00,16#00,16#00,16#00,16#00,16#00,16#00,16#00,16#9C,16#07,16#FC,16#1F,16#7C,16#3C,16#1C,16#38,16#1C,16#70,16#1C,16#70,16#1C,16#70,16#1C,16#70,16#1C,16#70,16#1C,16#70,16#3C,16#78,16#7C,16#38,16#DC,16#1F,16#1C,16#0F,16#1C,16#00,16#1C,16#00,16#1C,16#00,16#1C,16#00,16#1C,16#00,	// 16#71
16#00,16#00,16#00,16#00,16#00,16#00,16#00,16#00,16#00,16#00,16#00,16#00,16#00,16#00,16#7C,16#0E,16#FC,16#0E,16#8C,16#0F,16#0C,16#0F,16#00,16#0E,16#00,16#0E,16#00,16#0E,16#00,16#0E,16#00,16#0E,16#00,16#0E,16#00,16#0E,16#00,16#0E,16#00,16#0E,16#00,16#0E,16#00,16#00,16#00,16#00,16#00,16#00,16#00,16#00,16#00,16#00,	// 16#72
16#00,16#00,16#00,16#00,16#00,16#00,16#00,16#00,16#00,16#00,16#00,16#00,16#00,16#00,16#F0,16#07,16#F8,16#0F,16#08,16#1E,16#00,16#1C,16#00,16#1C,16#80,16#1F,16#E0,16#0F,16#F8,16#01,16#3C,16#00,16#1C,16#00,16#1C,16#00,16#3C,16#18,16#F8,16#1F,16#E0,16#0F,16#00,16#00,16#00,16#00,16#00,16#00,16#00,16#00,16#00,16#00,	// 16#73
16#00,16#00,16#00,16#00,16#00,16#00,16#00,16#00,16#00,16#00,16#00,16#07,16#00,16#07,16#FC,16#3F,16#FC,16#3F,16#00,16#07,16#00,16#07,16#00,16#07,16#00,16#07,16#00,16#07,16#00,16#07,16#00,16#07,16#00,16#07,16#00,16#07,16#80,16#07,16#FC,16#03,16#FC,16#01,16#00,16#00,16#00,16#00,16#00,16#00,16#00,16#00,16#00,16#00,	// 16#74
16#00,16#00,16#00,16#00,16#00,16#00,16#00,16#00,16#00,16#00,16#00,16#00,16#00,16#00,16#1C,16#38,16#1C,16#38,16#1C,16#38,16#1C,16#38,16#1C,16#38,16#1C,16#38,16#1C,16#38,16#1C,16#38,16#1C,16#38,16#1C,16#38,16#3C,16#38,16#7C,16#3C,16#DC,16#1F,16#1C,16#0F,16#00,16#00,16#00,16#00,16#00,16#00,16#00,16#00,16#00,16#00,	// 16#75
16#00,16#00,16#00,16#00,16#00,16#00,16#00,16#00,16#00,16#00,16#00,16#00,16#00,16#00,16#0E,16#78,16#1C,16#38,16#1C,16#38,16#1C,16#3C,16#18,16#1C,16#38,16#1C,16#38,16#0E,16#30,16#0E,16#70,16#07,16#70,16#07,16#60,16#07,16#E0,16#03,16#E0,16#03,16#C0,16#01,16#00,16#00,16#00,16#00,16#00,16#00,16#00,16#00,16#00,16#00,	// 16#76
16#00,16#00,16#00,16#00,16#00,16#00,16#00,16#00,16#00,16#00,16#00,16#00,16#00,16#00,16#03,16#C0,16#C3,16#E1,16#C2,16#E1,16#C6,16#63,16#C6,16#63,16#46,16#62,16#66,16#76,16#64,16#76,16#6C,16#36,16#6C,16#34,16#3C,16#3C,16#3C,16#3C,16#38,16#3C,16#38,16#18,16#00,16#00,16#00,16#00,16#00,16#00,16#00,16#00,16#00,16#00,	// 16#77
16#00,16#00,16#00,16#00,16#00,16#00,16#00,16#00,16#00,16#00,16#00,16#00,16#00,16#00,16#0C,16#78,16#18,16#3C,16#30,16#1E,16#70,16#0E,16#60,16#0F,16#C0,16#07,16#C0,16#03,16#C0,16#03,16#E0,16#07,16#F0,16#0E,16#70,16#0C,16#78,16#1C,16#3C,16#38,16#1E,16#70,16#00,16#00,16#00,16#00,16#00,16#00,16#00,16#00,16#00,16#00,	// 16#78
16#00,16#00,16#00,16#00,16#00,16#00,16#00,16#00,16#00,16#00,16#00,16#00,16#00,16#00,16#0E,16#78,16#0C,16#38,16#1C,16#38,16#18,16#1C,16#38,16#1C,16#38,16#1E,16#70,16#0E,16#70,16#0F,16#E0,16#07,16#E0,16#07,16#C0,16#03,16#C0,16#03,16#80,16#03,16#80,16#01,16#80,16#03,16#00,16#03,16#00,16#07,16#00,16#3E,16#00,16#3C,	// 16#79
16#00,16#00,16#00,16#00,16#00,16#00,16#00,16#00,16#00,16#00,16#00,16#00,16#00,16#00,16#FC,16#3F,16#FC,16#3F,16#1C,16#00,16#38,16#00,16#70,16#00,16#E0,16#00,16#C0,16#01,16#80,16#03,16#00,16#07,16#00,16#0E,16#00,16#1C,16#00,16#38,16#FC,16#3F,16#FC,16#3F,16#00,16#00,16#00,16#00,16#00,16#00,16#00,16#00,16#00,16#00,	// 16#7A
16#00,16#00,16#F8,16#00,16#F8,16#01,16#C0,16#03,16#80,16#03,16#80,16#03,16#80,16#03,16#C0,16#01,16#C0,16#01,16#C0,16#01,16#C0,16#01,16#80,16#03,16#00,16#1F,16#00,16#1F,16#80,16#03,16#C0,16#01,16#C0,16#01,16#C0,16#01,16#C0,16#01,16#80,16#03,16#80,16#03,16#80,16#03,16#C0,16#03,16#F8,16#01,16#F8,16#00,16#00,16#00,	// 16#7B
16#00,16#00,16#80,16#01,16#80,16#01,16#80,16#01,16#80,16#01,16#80,16#01,16#80,16#01,16#80,16#01,16#80,16#01,16#80,16#01,16#80,16#01,16#80,16#01,16#80,16#01,16#80,16#01,16#80,16#01,16#80,16#01,16#80,16#01,16#80,16#01,16#80,16#01,16#80,16#01,16#80,16#01,16#80,16#01,16#80,16#01,16#80,16#01,16#80,16#01,16#00,16#00,	// 16#7C
16#00,16#00,16#00,16#3E,16#00,16#3F,16#80,16#07,16#80,16#03,16#80,16#03,16#80,16#03,16#00,16#07,16#00,16#07,16#00,16#07,16#00,16#07,16#80,16#03,16#F0,16#01,16#F0,16#01,16#80,16#03,16#00,16#07,16#00,16#07,16#00,16#07,16#00,16#07,16#80,16#03,16#80,16#03,16#80,16#03,16#80,16#07,16#00,16#3F,16#00,16#3E,16#00,16#00,	// 16#7D
16#00,16#00,16#00,16#00,16#00,16#00,16#00,16#00,16#00,16#00,16#00,16#00,16#00,16#00,16#00,16#00,16#00,16#00,16#00,16#00,16#00,16#00,16#00,16#00,16#06,16#1E,16#C6,16#3F,16#FC,16#63,16#78,16#60,16#00,16#00,16#00,16#00,16#00,16#00,16#00,16#00,16#00,16#00,16#00,16#00,16#00,16#00,16#00,16#00,16#00,16#00,16#00,16#00,	// 16#7E
16#00,16#00,16#00,16#00,16#00,16#00,16#00,16#00,16#00,16#00,16#F0,16#1F,16#10,16#10,16#10,16#10,16#10,16#10,16#10,16#10,16#10,16#10,16#10,16#10,16#10,16#10,16#10,16#10,16#10,16#10,16#10,16#10,16#10,16#10,16#10,16#10,16#10,16#10,16#10,16#10,16#F0,16#1F,16#00,16#00,16#00,16#00,16#00,16#00,16#00,16#00,16#00,16#00,	// 16#7F
16#00,16#00,16#00,16#00,16#00,16#00,16#00,16#00,16#00,16#00,16#F8,16#03,16#FC,16#0F,16#0C,16#1E,16#00,16#3C,16#00,16#38,16#00,16#70,16#00,16#70,16#00,16#70,16#00,16#70,16#00,16#70,16#00,16#70,16#00,16#38,16#00,16#3C,16#04,16#1E,16#FC,16#0F,16#F8,16#03,16#40,16#00,16#E0,16#00,16#30,16#00,16#30,16#00,16#E0,16#01,	// 16#80
16#00,16#00,16#00,16#00,16#00,16#00,16#60,16#0C,16#60,16#0C,16#00,16#00,16#00,16#00,16#1C,16#38,16#1C,16#38,16#1C,16#38,16#1C,16#38,16#1C,16#38,16#1C,16#38,16#1C,16#38,16#1C,16#38,16#1C,16#38,16#1C,16#38,16#3C,16#38,16#7C,16#3C,16#DC,16#1F,16#1C,16#0F,16#00,16#00,16#00,16#00,16#00,16#00,16#00,16#00,16#00,16#00,	// 16#81
16#00,16#00,16#30,16#00,16#60,16#00,16#C0,16#00,16#80,16#01,16#00,16#00,16#00,16#00,16#E0,16#03,16#F0,16#0F,16#38,16#1E,16#1C,16#1C,16#1C,16#38,16#1C,16#38,16#FC,16#3F,16#FC,16#3F,16#00,16#38,16#00,16#38,16#00,16#1C,16#04,16#1E,16#FC,16#0F,16#F8,16#03,16#00,16#00,16#00,16#00,16#00,16#00,16#00,16#00,16#00,16#00,	// 16#82
16#00,16#00,16#80,16#03,16#C0,16#06,16#60,16#0C,16#30,16#18,16#00,16#00,16#00,16#00,16#E0,16#07,16#F0,16#1F,16#78,16#18,16#38,16#00,16#38,16#00,16#F8,16#07,16#F8,16#0F,16#38,16#1C,16#38,16#38,16#38,16#38,16#38,16#38,16#78,16#3C,16#DE,16#1F,16#1E,16#0F,16#00,16#00,16#00,16#00,16#00,16#00,16#00,16#00,16#00,16#00,	// 16#83
16#00,16#00,16#00,16#00,16#00,16#00,16#30,16#06,16#30,16#06,16#00,16#00,16#00,16#00,16#E0,16#07,16#F0,16#1F,16#78,16#18,16#38,16#00,16#38,16#00,16#F8,16#07,16#F8,16#0F,16#38,16#1C,16#38,16#38,16#38,16#38,16#38,16#38,16#78,16#3C,16#DE,16#1F,16#1E,16#0F,16#00,16#00,16#00,16#00,16#00,16#00,16#00,16#00,16#00,16#00,	// 16#84
16#00,16#00,16#00,16#0C,16#00,16#06,16#00,16#03,16#80,16#01,16#00,16#00,16#00,16#00,16#E0,16#07,16#F0,16#1F,16#78,16#18,16#38,16#00,16#38,16#00,16#F8,16#07,16#F8,16#0F,16#38,16#1C,16#38,16#38,16#38,16#38,16#38,16#38,16#78,16#3C,16#DE,16#1F,16#1E,16#0F,16#00,16#00,16#00,16#00,16#00,16#00,16#00,16#00,16#00,16#00,	// 16#85
16#80,16#03,16#40,16#04,16#40,16#04,16#40,16#04,16#80,16#03,16#00,16#00,16#00,16#00,16#E0,16#07,16#F0,16#1F,16#78,16#18,16#38,16#00,16#38,16#00,16#F8,16#07,16#F8,16#0F,16#38,16#1C,16#38,16#38,16#38,16#38,16#38,16#38,16#78,16#3C,16#DE,16#1F,16#1E,16#0F,16#00,16#00,16#00,16#00,16#00,16#00,16#00,16#00,16#00,16#00,	// 16#86
16#00,16#00,16#00,16#00,16#00,16#00,16#00,16#00,16#00,16#00,16#00,16#00,16#00,16#00,16#F8,16#03,16#FC,16#0F,16#04,16#1E,16#00,16#1C,16#00,16#38,16#00,16#38,16#00,16#38,16#00,16#38,16#00,16#38,16#00,16#3C,16#00,16#1C,16#04,16#1F,16#FC,16#0F,16#F8,16#03,16#80,16#00,16#C0,16#01,16#60,16#00,16#60,16#00,16#C0,16#03,	// 16#87
16#00,16#00,16#80,16#03,16#C0,16#06,16#60,16#0C,16#30,16#18,16#00,16#00,16#00,16#00,16#E0,16#03,16#F0,16#0F,16#38,16#1E,16#1C,16#1C,16#1C,16#38,16#1C,16#38,16#FC,16#3F,16#FC,16#3F,16#00,16#38,16#00,16#38,16#00,16#1C,16#04,16#1E,16#FC,16#0F,16#F8,16#03,16#00,16#00,16#00,16#00,16#00,16#00,16#00,16#00,16#00,16#00,	// 16#88
16#00,16#00,16#00,16#00,16#00,16#00,16#30,16#06,16#30,16#06,16#00,16#00,16#00,16#00,16#E0,16#03,16#F0,16#0F,16#38,16#1E,16#1C,16#1C,16#1C,16#38,16#1C,16#38,16#FC,16#3F,16#FC,16#3F,16#00,16#38,16#00,16#38,16#00,16#1C,16#04,16#1E,16#FC,16#0F,16#F8,16#03,16#00,16#00,16#00,16#00,16#00,16#00,16#00,16#00,16#00,16#00,	// 16#89
16#00,16#00,16#00,16#0C,16#00,16#06,16#00,16#03,16#80,16#01,16#00,16#00,16#00,16#00,16#E0,16#03,16#F0,16#0F,16#38,16#1E,16#1C,16#1C,16#1C,16#38,16#1C,16#38,16#FC,16#3F,16#FC,16#3F,16#00,16#38,16#00,16#38,16#00,16#1C,16#04,16#1E,16#FC,16#0F,16#F8,16#03,16#00,16#00,16#00,16#00,16#00,16#00,16#00,16#00,16#00,16#00,	// 16#8A
16#00,16#00,16#00,16#00,16#00,16#00,16#60,16#0C,16#60,16#0C,16#00,16#00,16#00,16#00,16#C0,16#3F,16#C0,16#3F,16#C0,16#01,16#C0,16#01,16#C0,16#01,16#C0,16#01,16#C0,16#01,16#C0,16#01,16#C0,16#01,16#C0,16#01,16#C0,16#01,16#C0,16#01,16#C0,16#01,16#C0,16#01,16#00,16#00,16#00,16#00,16#00,16#00,16#00,16#00,16#00,16#00,	// 16#8B
16#00,16#00,16#C0,16#01,16#60,16#03,16#30,16#06,16#18,16#0C,16#00,16#00,16#00,16#00,16#C0,16#3F,16#C0,16#3F,16#C0,16#01,16#C0,16#01,16#C0,16#01,16#C0,16#01,16#C0,16#01,16#C0,16#01,16#C0,16#01,16#C0,16#01,16#C0,16#01,16#C0,16#01,16#C0,16#01,16#C0,16#01,16#00,16#00,16#00,16#00,16#00,16#00,16#00,16#00,16#00,16#00,	// 16#8C
16#00,16#00,16#00,16#06,16#00,16#03,16#80,16#01,16#C0,16#00,16#00,16#00,16#00,16#00,16#C0,16#3F,16#C0,16#3F,16#C0,16#01,16#C0,16#01,16#C0,16#01,16#C0,16#01,16#C0,16#01,16#C0,16#01,16#C0,16#01,16#C0,16#01,16#C0,16#01,16#C0,16#01,16#C0,16#01,16#C0,16#01,16#00,16#00,16#00,16#00,16#00,16#00,16#00,16#00,16#00,16#00,	// 16#8D
16#30,16#0C,16#30,16#0C,16#00,16#00,16#00,16#00,16#00,16#00,16#80,16#03,16#C0,16#03,16#C0,16#07,16#E0,16#06,16#E0,16#06,16#60,16#0E,16#70,16#0C,16#70,16#1C,16#38,16#1C,16#38,16#18,16#FC,16#3F,16#FC,16#3F,16#1C,16#70,16#0E,16#70,16#0E,16#70,16#07,16#E0,16#00,16#00,16#00,16#00,16#00,16#00,16#00,16#00,16#00,16#00,	// 16#8E
16#C0,16#01,16#20,16#02,16#20,16#02,16#20,16#02,16#C0,16#01,16#C0,16#01,16#E0,16#03,16#E0,16#03,16#60,16#07,16#70,16#06,16#70,16#06,16#30,16#0E,16#38,16#0C,16#38,16#1C,16#1C,16#1C,16#FC,16#3F,16#FC,16#3F,16#0E,16#38,16#0E,16#70,16#0E,16#70,16#07,16#E0,16#00,16#00,16#00,16#00,16#00,16#00,16#00,16#00,16#00,16#00,	// 16#8F
16#70,16#00,16#E0,16#00,16#C0,16#01,16#00,16#00,16#00,16#00,16#FC,16#1F,16#FC,16#1F,16#00,16#1C,16#00,16#1C,16#00,16#1C,16#00,16#1C,16#00,16#1C,16#F8,16#1F,16#F8,16#1F,16#00,16#1C,16#00,16#1C,16#00,16#1C,16#00,16#1C,16#00,16#1C,16#FE,16#1F,16#FE,16#1F,16#00,16#00,16#00,16#00,16#00,16#00,16#00,16#00,16#00,16#00,	// 16#90
16#00,16#00,16#00,16#00,16#00,16#00,16#00,16#00,16#00,16#00,16#00,16#00,16#00,16#00,16#3C,16#1F,16#FE,16#3F,16#E6,16#01,16#C7,16#01,16#C7,16#01,16#FF,16#0F,16#FF,16#3F,16#C0,16#39,16#C0,16#71,16#C0,16#71,16#C0,16#71,16#E1,16#79,16#FF,16#3F,16#3E,16#1E,16#00,16#00,16#00,16#00,16#00,16#00,16#00,16#00,16#00,16#00,	// 16#91
16#00,16#00,16#00,16#00,16#00,16#00,16#00,16#00,16#00,16#00,16#FC,16#01,16#FC,16#03,16#E0,16#03,16#E0,16#07,16#E0,16#06,16#E0,16#06,16#E0,16#0E,16#FC,16#0C,16#FC,16#1C,16#E0,16#18,16#E0,16#38,16#E0,16#3F,16#E0,16#3F,16#E0,16#60,16#FE,16#60,16#FE,16#C0,16#00,16#00,16#00,16#00,16#00,16#00,16#00,16#00,16#00,16#00,	// 16#92
16#00,16#00,16#80,16#03,16#C0,16#06,16#60,16#0C,16#30,16#18,16#00,16#00,16#00,16#00,16#C0,16#07,16#F0,16#1F,16#78,16#3C,16#38,16#38,16#1C,16#70,16#1C,16#70,16#1C,16#70,16#1C,16#70,16#1C,16#70,16#1C,16#70,16#38,16#38,16#78,16#3C,16#F0,16#1F,16#C0,16#07,16#00,16#00,16#00,16#00,16#00,16#00,16#00,16#00,16#00,16#00,	// 16#93
16#00,16#00,16#00,16#00,16#00,16#00,16#60,16#0C,16#60,16#0C,16#00,16#00,16#00,16#00,16#C0,16#07,16#F0,16#1F,16#78,16#3C,16#38,16#38,16#1C,16#70,16#1C,16#70,16#1C,16#70,16#1C,16#70,16#1C,16#70,16#1C,16#70,16#38,16#38,16#78,16#3C,16#F0,16#1F,16#C0,16#07,16#00,16#00,16#00,16#00,16#00,16#00,16#00,16#00,16#00,16#00,	// 16#94
16#00,16#00,16#00,16#0C,16#00,16#06,16#00,16#03,16#80,16#01,16#00,16#00,16#00,16#00,16#C0,16#07,16#F0,16#1F,16#78,16#3C,16#38,16#38,16#1C,16#70,16#1C,16#70,16#1C,16#70,16#1C,16#70,16#1C,16#70,16#1C,16#70,16#38,16#38,16#78,16#3C,16#F0,16#1F,16#C0,16#07,16#00,16#00,16#00,16#00,16#00,16#00,16#00,16#00,16#00,16#00,	// 16#95
16#00,16#00,16#80,16#03,16#C0,16#06,16#60,16#0C,16#30,16#18,16#00,16#00,16#00,16#00,16#1C,16#38,16#1C,16#38,16#1C,16#38,16#1C,16#38,16#1C,16#38,16#1C,16#38,16#1C,16#38,16#1C,16#38,16#1C,16#38,16#1C,16#38,16#3C,16#38,16#7C,16#3C,16#DC,16#1F,16#1C,16#0F,16#00,16#00,16#00,16#00,16#00,16#00,16#00,16#00,16#00,16#00,	// 16#96
16#00,16#00,16#00,16#0C,16#00,16#06,16#00,16#03,16#80,16#01,16#00,16#00,16#00,16#00,16#1C,16#38,16#1C,16#38,16#1C,16#38,16#1C,16#38,16#1C,16#38,16#1C,16#38,16#1C,16#38,16#1C,16#38,16#1C,16#38,16#1C,16#38,16#3C,16#38,16#7C,16#3C,16#DC,16#1F,16#1C,16#0F,16#00,16#00,16#00,16#00,16#00,16#00,16#00,16#00,16#00,16#00,	// 16#97
16#00,16#00,16#00,16#00,16#00,16#00,16#60,16#0C,16#60,16#0C,16#00,16#00,16#00,16#00,16#0E,16#78,16#0C,16#38,16#1C,16#38,16#18,16#1C,16#38,16#1C,16#38,16#1E,16#70,16#0E,16#70,16#0F,16#E0,16#07,16#E0,16#07,16#C0,16#03,16#C0,16#03,16#80,16#03,16#80,16#01,16#80,16#03,16#00,16#03,16#00,16#07,16#00,16#3E,16#00,16#3C,	// 16#98
16#30,16#0C,16#30,16#0C,16#00,16#00,16#00,16#00,16#00,16#00,16#E0,16#07,16#F0,16#0F,16#38,16#1C,16#1C,16#38,16#1C,16#38,16#0E,16#70,16#0E,16#70,16#0E,16#70,16#0E,16#70,16#0E,16#70,16#0E,16#70,16#1C,16#38,16#1C,16#38,16#38,16#1C,16#F0,16#0F,16#E0,16#07,16#00,16#00,16#00,16#00,16#00,16#00,16#00,16#00,16#00,16#00,	// 16#99
16#18,16#06,16#18,16#06,16#00,16#00,16#00,16#00,16#00,16#00,16#0E,16#38,16#0E,16#38,16#0E,16#38,16#0E,16#38,16#0E,16#38,16#0E,16#38,16#0E,16#38,16#0E,16#38,16#0E,16#38,16#0E,16#38,16#0E,16#38,16#0E,16#38,16#1E,16#3C,16#1C,16#1C,16#F8,16#0F,16#F0,16#07,16#00,16#00,16#00,16#00,16#00,16#00,16#00,16#00,16#00,16#00,	// 16#9A
16#00,16#00,16#00,16#00,16#00,16#00,16#00,16#00,16#00,16#00,16#00,16#00,16#00,16#00,16#CC,16#07,16#F8,16#1F,16#78,16#3C,16#78,16#38,16#DC,16#70,16#9C,16#70,16#9C,16#71,16#1C,16#73,16#1C,16#76,16#1C,16#76,16#38,16#3C,16#78,16#3C,16#F0,16#3F,16#C0,16#67,16#00,16#00,16#00,16#00,16#00,16#00,16#00,16#00,16#00,16#00,	// 16#9B
16#00,16#00,16#00,16#00,16#7C,16#00,16#FC,16#01,16#C0,16#01,16#80,16#03,16#80,16#03,16#80,16#03,16#80,16#03,16#80,16#03,16#F0,16#0F,16#F0,16#0F,16#80,16#03,16#80,16#03,16#80,16#03,16#80,16#03,16#00,16#07,16#00,16#0E,16#FC,16#1F,16#FC,16#1F,16#FC,16#1F,16#00,16#00,16#00,16#00,16#00,16#00,16#00,16#00,16#00,16#00,	// 16#9C
16#00,16#00,16#00,16#00,16#00,16#00,16#00,16#00,16#00,16#00,16#E6,16#07,16#FC,16#0F,16#38,16#1C,16#3C,16#38,16#3C,16#38,16#6E,16#70,16#CE,16#70,16#8E,16#71,16#8E,16#71,16#0E,16#73,16#0E,16#76,16#1C,16#3C,16#1C,16#3C,16#38,16#1C,16#F0,16#3F,16#E0,16#67,16#00,16#00,16#00,16#00,16#00,16#00,16#00,16#00,16#00,16#00,	// 16#9D
16#00,16#00,16#00,16#00,16#00,16#00,16#00,16#00,16#00,16#00,16#00,16#00,16#00,16#00,16#04,16#20,16#0E,16#70,16#1C,16#38,16#38,16#1C,16#70,16#0E,16#E0,16#07,16#C0,16#03,16#C0,16#03,16#E0,16#07,16#70,16#0E,16#38,16#1C,16#1C,16#38,16#0E,16#70,16#04,16#20,16#00,16#00,16#00,16#00,16#00,16#00,16#00,16#00,16#00,16#00,	// 16#9E
16#00,16#00,16#FC,16#00,16#FC,16#01,16#80,16#03,16#80,16#03,16#80,16#03,16#80,16#03,16#F8,16#1F,16#F8,16#1F,16#80,16#03,16#80,16#03,16#80,16#03,16#80,16#03,16#80,16#03,16#80,16#03,16#80,16#03,16#80,16#03,16#80,16#03,16#80,16#03,16#80,16#03,16#80,16#03,16#80,16#03,16#80,16#03,16#80,16#03,16#00,16#7F,16#00,16#7E,	// 16#9F
16#00,16#00,16#60,16#00,16#C0,16#00,16#80,16#01,16#00,16#03,16#00,16#00,16#00,16#00,16#E0,16#07,16#F0,16#1F,16#78,16#18,16#38,16#00,16#38,16#00,16#F8,16#07,16#F8,16#0F,16#38,16#1C,16#38,16#38,16#38,16#38,16#38,16#38,16#78,16#3C,16#DE,16#1F,16#1E,16#0F,16#00,16#00,16#00,16#00,16#00,16#00,16#00,16#00,16#00,16#00,	// 16#A0
16#00,16#00,16#60,16#00,16#C0,16#00,16#80,16#01,16#00,16#03,16#00,16#00,16#00,16#00,16#C0,16#3F,16#C0,16#3F,16#C0,16#01,16#C0,16#01,16#C0,16#01,16#C0,16#01,16#C0,16#01,16#C0,16#01,16#C0,16#01,16#C0,16#01,16#C0,16#01,16#C0,16#01,16#C0,16#01,16#C0,16#01,16#00,16#00,16#00,16#00,16#00,16#00,16#00,16#00,16#00,16#00,	// 16#A1
16#00,16#00,16#60,16#00,16#C0,16#00,16#80,16#01,16#00,16#03,16#00,16#00,16#00,16#00,16#C0,16#07,16#F0,16#1F,16#78,16#3C,16#38,16#38,16#1C,16#70,16#1C,16#70,16#1C,16#70,16#1C,16#70,16#1C,16#70,16#1C,16#70,16#38,16#38,16#78,16#3C,16#F0,16#1F,16#C0,16#07,16#00,16#00,16#00,16#00,16#00,16#00,16#00,16#00,16#00,16#00,	// 16#A2
16#00,16#00,16#60,16#00,16#C0,16#00,16#80,16#01,16#00,16#03,16#00,16#00,16#00,16#00,16#1C,16#38,16#1C,16#38,16#1C,16#38,16#1C,16#38,16#1C,16#38,16#1C,16#38,16#1C,16#38,16#1C,16#38,16#1C,16#38,16#1C,16#38,16#3C,16#38,16#7C,16#3C,16#DC,16#1F,16#1C,16#0F,16#00,16#00,16#00,16#00,16#00,16#00,16#00,16#00,16#00,16#00,	// 16#A3
16#00,16#00,16#00,16#00,16#30,16#07,16#F0,16#0F,16#E0,16#0C,16#00,16#00,16#00,16#00,16#F0,16#38,16#F8,16#3B,16#3C,16#3E,16#1C,16#3C,16#1C,16#38,16#1C,16#38,16#1C,16#38,16#1C,16#38,16#1C,16#38,16#1C,16#38,16#1C,16#38,16#1C,16#38,16#1C,16#38,16#1C,16#38,16#00,16#00,16#00,16#00,16#00,16#00,16#00,16#00,16#00,16#00,	// 16#A4
16#30,16#07,16#F0,16#0F,16#E0,16#0C,16#00,16#00,16#00,16#00,16#0C,16#38,16#0C,16#38,16#0C,16#3C,16#0C,16#3E,16#0C,16#3E,16#0C,16#3F,16#8C,16#37,16#8C,16#33,16#CC,16#33,16#EC,16#31,16#FC,16#30,16#7C,16#30,16#7C,16#30,16#3C,16#30,16#1C,16#30,16#1C,16#30,16#00,16#00,16#00,16#00,16#00,16#00,16#00,16#00,16#00,16#00,	// 16#A5
16#00,16#00,16#00,16#00,16#C0,16#07,16#E0,16#0F,16#60,16#08,16#E0,16#07,16#E0,16#0F,16#60,16#1C,16#60,16#18,16#E0,16#18,16#F8,16#1F,16#38,16#0F,16#00,16#00,16#00,16#00,16#00,16#00,16#00,16#00,16#00,16#00,16#00,16#00,16#00,16#00,16#00,16#00,16#00,16#00,16#00,16#00,16#00,16#00,16#00,16#00,16#00,16#00,16#00,16#00,	// 16#A6
16#00,16#00,16#00,16#00,16#E0,16#07,16#F0,16#0F,16#38,16#1C,16#18,16#18,16#18,16#18,16#18,16#18,16#18,16#18,16#38,16#1C,16#F0,16#0F,16#E0,16#07,16#00,16#00,16#00,16#00,16#00,16#00,16#00,16#00,16#00,16#00,16#00,16#00,16#00,16#00,16#00,16#00,16#00,16#00,16#00,16#00,16#00,16#00,16#00,16#00,16#00,16#00,16#00,16#00,	// 16#A7
16#00,16#00,16#00,16#00,16#00,16#00,16#00,16#00,16#00,16#00,16#00,16#00,16#00,16#00,16#C0,16#01,16#C0,16#01,16#C0,16#01,16#00,16#00,16#00,16#00,16#C0,16#01,16#C0,16#01,16#C0,16#01,16#80,16#03,16#80,16#07,16#00,16#0F,16#00,16#1E,16#00,16#1C,16#00,16#38,16#00,16#38,16#0C,16#38,16#0C,16#3C,16#FC,16#1F,16#F8,16#07,	// 16#A8
16#00,16#00,16#00,16#00,16#C0,16#07,16#20,16#08,16#90,16#17,16#48,16#24,16#48,16#24,16#88,16#27,16#88,16#24,16#88,16#24,16#D0,16#14,16#20,16#08,16#C0,16#07,16#00,16#00,16#00,16#00,16#00,16#00,16#00,16#00,16#00,16#00,16#00,16#00,16#00,16#00,16#00,16#00,16#00,16#00,16#00,16#00,16#00,16#00,16#00,16#00,16#00,16#00,	// 16#A9
16#00,16#00,16#00,16#00,16#00,16#00,16#00,16#00,16#00,16#00,16#00,16#00,16#00,16#00,16#00,16#00,16#00,16#00,16#00,16#00,16#00,16#00,16#FE,16#7F,16#FE,16#7F,16#06,16#00,16#06,16#00,16#06,16#00,16#06,16#00,16#00,16#00,16#00,16#00,16#00,16#00,16#00,16#00,16#00,16#00,16#00,16#00,16#00,16#00,16#00,16#00,16#00,16#00,	// 16#AA
16#00,16#00,16#00,16#00,16#30,16#F8,16#60,16#F8,16#60,16#38,16#C0,16#38,16#C0,16#38,16#80,16#39,16#80,16#39,16#00,16#3B,16#00,16#3B,16#3C,16#3E,16#7F,16#0C,16#07,16#0C,16#07,16#18,16#0E,16#18,16#1C,16#30,16#30,16#30,16#60,16#60,16#7F,16#60,16#7F,16#C0,16#00,16#00,16#00,16#00,16#00,16#00,16#00,16#00,16#00,16#00,	// 16#AB
16#00,16#00,16#00,16#00,16#18,16#F8,16#30,16#F8,16#30,16#38,16#60,16#38,16#60,16#38,16#C0,16#38,16#C0,16#38,16#80,16#39,16#80,16#39,16#1C,16#3B,16#3C,16#06,16#5C,16#06,16#9C,16#0C,16#9C,16#0D,16#1C,16#1B,16#FF,16#1B,16#1C,16#30,16#1C,16#30,16#1C,16#60,16#00,16#00,16#00,16#00,16#00,16#00,16#00,16#00,16#00,16#00,	// 16#AC
16#00,16#00,16#00,16#00,16#00,16#00,16#00,16#00,16#00,16#00,16#00,16#00,16#00,16#00,16#80,16#03,16#80,16#03,16#80,16#03,16#00,16#00,16#00,16#00,16#80,16#03,16#80,16#03,16#80,16#03,16#80,16#03,16#80,16#03,16#80,16#03,16#80,16#03,16#80,16#03,16#80,16#03,16#80,16#03,16#80,16#03,16#80,16#03,16#80,16#03,16#80,16#03,	// 16#AD
16#00,16#00,16#00,16#00,16#00,16#00,16#00,16#00,16#00,16#00,16#00,16#00,16#00,16#00,16#00,16#00,16#08,16#02,16#1C,16#07,16#38,16#0E,16#70,16#1C,16#E0,16#38,16#C0,16#30,16#C0,16#71,16#E0,16#38,16#70,16#1C,16#38,16#0E,16#1C,16#07,16#08,16#02,16#00,16#00,16#00,16#00,16#00,16#00,16#00,16#00,16#00,16#00,16#00,16#00,	// 16#AE
16#00,16#00,16#00,16#00,16#00,16#00,16#00,16#00,16#00,16#00,16#00,16#00,16#00,16#00,16#00,16#00,16#80,16#10,16#C0,16#39,16#E0,16#1C,16#70,16#0E,16#38,16#07,16#9C,16#03,16#18,16#03,16#38,16#07,16#70,16#0E,16#E0,16#1C,16#C0,16#39,16#80,16#10,16#00,16#00,16#00,16#00,16#00,16#00,16#00,16#00,16#00,16#00,16#00,16#00,	// 16#AF
16#38,16#E7,16#38,16#E7,16#38,16#E7,16#00,16#00,16#00,16#00,16#38,16#E7,16#38,16#E7,16#38,16#E7,16#00,16#00,16#00,16#00,16#38,16#E7,16#38,16#E7,16#38,16#E7,16#00,16#00,16#00,16#00,16#00,16#00,16#38,16#E7,16#38,16#E7,16#38,16#E7,16#00,16#00,16#00,16#00,16#38,16#E7,16#38,16#E7,16#38,16#E7,16#00,16#00,16#00,16#00,	// 16#B0
16#E7,16#1C,16#E7,16#1C,16#E7,16#1C,16#38,16#E7,16#38,16#E7,16#FF,16#FF,16#E7,16#1C,16#E7,16#1C,16#38,16#E7,16#38,16#E7,16#FF,16#FF,16#E7,16#1C,16#E7,16#1C,16#38,16#E7,16#38,16#E7,16#38,16#E7,16#E7,16#1C,16#E7,16#1C,16#FF,16#FF,16#38,16#E7,16#38,16#E7,16#E7,16#1C,16#E7,16#1C,16#FF,16#FF,16#38,16#E7,16#38,16#E7,	// 16#B1
16#FF,16#FF,16#FF,16#FF,16#FF,16#FF,16#38,16#E7,16#38,16#E7,16#FF,16#FF,16#FF,16#FF,16#FF,16#FF,16#38,16#E7,16#38,16#E7,16#FF,16#FF,16#FF,16#FF,16#FF,16#FF,16#38,16#E7,16#38,16#E7,16#38,16#E7,16#FF,16#FF,16#FF,16#FF,16#FF,16#FF,16#38,16#E7,16#38,16#E7,16#FF,16#FF,16#FF,16#FF,16#FF,16#FF,16#38,16#E7,16#38,16#E7,	// 16#B2
16#80,16#01,16#80,16#01,16#80,16#01,16#80,16#01,16#80,16#01,16#80,16#01,16#80,16#01,16#80,16#01,16#80,16#01,16#80,16#01,16#80,16#01,16#80,16#01,16#80,16#01,16#80,16#01,16#80,16#01,16#80,16#01,16#80,16#01,16#80,16#01,16#80,16#01,16#80,16#01,16#80,16#01,16#80,16#01,16#80,16#01,16#80,16#01,16#80,16#01,16#80,16#01,	// 16#B3
16#80,16#01,16#80,16#01,16#80,16#01,16#80,16#01,16#80,16#01,16#80,16#01,16#80,16#01,16#80,16#01,16#80,16#01,16#80,16#01,16#80,16#01,16#80,16#01,16#80,16#FF,16#80,16#FF,16#80,16#01,16#80,16#01,16#80,16#01,16#80,16#01,16#80,16#01,16#80,16#01,16#80,16#01,16#80,16#01,16#80,16#01,16#80,16#01,16#80,16#01,16#80,16#01,	// 16#B4
16#E0,16#00,16#C0,16#01,16#80,16#03,16#00,16#00,16#00,16#00,16#80,16#03,16#C0,16#03,16#C0,16#07,16#E0,16#06,16#E0,16#06,16#60,16#0E,16#70,16#0C,16#70,16#1C,16#38,16#1C,16#38,16#18,16#FC,16#3F,16#FC,16#3F,16#1C,16#70,16#0E,16#70,16#0E,16#70,16#07,16#E0,16#00,16#00,16#00,16#00,16#00,16#00,16#00,16#00,16#00,16#00,	// 16#B5
16#C0,16#07,16#E0,16#0E,16#70,16#1C,16#00,16#00,16#00,16#00,16#80,16#03,16#C0,16#03,16#C0,16#07,16#E0,16#06,16#E0,16#06,16#60,16#0E,16#70,16#0C,16#70,16#1C,16#38,16#1C,16#38,16#18,16#FC,16#3F,16#FC,16#3F,16#1C,16#70,16#0E,16#70,16#0E,16#70,16#07,16#E0,16#00,16#00,16#00,16#00,16#00,16#00,16#00,16#00,16#00,16#00,	// 16#B6
16#00,16#07,16#80,16#03,16#C0,16#01,16#00,16#00,16#00,16#00,16#80,16#03,16#C0,16#03,16#C0,16#07,16#E0,16#06,16#E0,16#06,16#60,16#0E,16#70,16#0C,16#70,16#1C,16#38,16#1C,16#38,16#18,16#FC,16#3F,16#FC,16#3F,16#1C,16#70,16#0E,16#70,16#0E,16#70,16#07,16#E0,16#00,16#00,16#00,16#00,16#00,16#00,16#00,16#00,16#00,16#00,	// 16#B7
16#00,16#00,16#00,16#00,16#F0,16#07,16#F8,16#0F,16#1C,16#1C,16#0E,16#38,16#F6,16#31,16#F7,16#77,16#13,16#66,16#03,16#6C,16#03,16#6C,16#03,16#6C,16#03,16#6C,16#03,16#6C,16#13,16#66,16#F7,16#77,16#E6,16#31,16#0E,16#38,16#1C,16#1C,16#F8,16#0F,16#F0,16#07,16#00,16#00,16#00,16#00,16#00,16#00,16#00,16#00,16#00,16#00,	// 16#B8
16#60,16#06,16#60,16#06,16#60,16#06,16#60,16#06,16#60,16#06,16#60,16#06,16#60,16#06,16#60,16#06,16#60,16#06,16#60,16#06,16#60,16#FE,16#60,16#FE,16#60,16#00,16#60,16#00,16#60,16#FE,16#60,16#FE,16#60,16#06,16#60,16#06,16#60,16#06,16#60,16#06,16#60,16#06,16#60,16#06,16#60,16#06,16#60,16#06,16#60,16#06,16#60,16#06,	// 16#B9
16#60,16#06,16#60,16#06,16#60,16#06,16#60,16#06,16#60,16#06,16#60,16#06,16#60,16#06,16#60,16#06,16#60,16#06,16#60,16#06,16#60,16#06,16#60,16#06,16#60,16#06,16#60,16#06,16#60,16#06,16#60,16#06,16#60,16#06,16#60,16#06,16#60,16#06,16#60,16#06,16#60,16#06,16#60,16#06,16#60,16#06,16#60,16#06,16#60,16#06,16#60,16#06,	// 16#BA
16#00,16#00,16#00,16#00,16#00,16#00,16#00,16#00,16#00,16#00,16#00,16#00,16#00,16#00,16#00,16#00,16#00,16#00,16#00,16#00,16#E0,16#FF,16#E0,16#FF,16#60,16#00,16#60,16#00,16#60,16#FE,16#60,16#FE,16#60,16#06,16#60,16#06,16#60,16#06,16#60,16#06,16#60,16#06,16#60,16#06,16#60,16#06,16#60,16#06,16#60,16#06,16#60,16#06,	// 16#BB
16#60,16#06,16#60,16#06,16#60,16#06,16#60,16#06,16#60,16#06,16#60,16#06,16#60,16#06,16#60,16#06,16#60,16#06,16#60,16#06,16#60,16#FE,16#60,16#FE,16#60,16#00,16#60,16#00,16#E0,16#FF,16#E0,16#FF,16#00,16#00,16#00,16#00,16#00,16#00,16#00,16#00,16#00,16#00,16#00,16#00,16#00,16#00,16#00,16#00,16#00,16#00,16#00,16#00,	// 16#BC
16#00,16#00,16#00,16#00,16#80,16#01,16#80,16#01,16#F0,16#03,16#F0,16#0F,16#90,16#1D,16#80,16#1D,16#80,16#39,16#80,16#39,16#80,16#39,16#80,16#39,16#80,16#39,16#80,16#39,16#80,16#39,16#80,16#1D,16#90,16#1F,16#F0,16#0F,16#E0,16#07,16#80,16#01,16#80,16#01,16#00,16#00,16#00,16#00,16#00,16#00,16#00,16#00,16#00,16#00,	// 16#BD
16#00,16#00,16#00,16#00,16#07,16#70,16#06,16#38,16#0C,16#1C,16#0C,16#1C,16#18,16#0E,16#30,16#07,16#30,16#07,16#E0,16#03,16#C0,16#01,16#FC,16#1F,16#FC,16#1F,16#C0,16#01,16#C0,16#01,16#C0,16#01,16#FC,16#1F,16#FC,16#1F,16#C0,16#01,16#C0,16#01,16#C0,16#01,16#00,16#00,16#00,16#00,16#00,16#00,16#00,16#00,16#00,16#00,	// 16#BE
16#00,16#00,16#00,16#00,16#00,16#00,16#00,16#00,16#00,16#00,16#00,16#00,16#00,16#00,16#00,16#00,16#00,16#00,16#00,16#00,16#00,16#00,16#00,16#00,16#80,16#FF,16#80,16#FF,16#80,16#01,16#80,16#01,16#80,16#01,16#80,16#01,16#80,16#01,16#80,16#01,16#80,16#01,16#80,16#01,16#80,16#01,16#80,16#01,16#80,16#01,16#80,16#01,	// 16#BF
16#80,16#01,16#80,16#01,16#80,16#01,16#80,16#01,16#80,16#01,16#80,16#01,16#80,16#01,16#80,16#01,16#80,16#01,16#80,16#01,16#80,16#01,16#80,16#01,16#FF,16#01,16#FF,16#01,16#00,16#00,16#00,16#00,16#00,16#00,16#00,16#00,16#00,16#00,16#00,16#00,16#00,16#00,16#00,16#00,16#00,16#00,16#00,16#00,16#00,16#00,16#00,16#00,	// 16#C0
16#80,16#01,16#80,16#01,16#80,16#01,16#80,16#01,16#80,16#01,16#80,16#01,16#80,16#01,16#80,16#01,16#80,16#01,16#80,16#01,16#80,16#01,16#80,16#01,16#FF,16#FF,16#FF,16#FF,16#00,16#00,16#00,16#00,16#00,16#00,16#00,16#00,16#00,16#00,16#00,16#00,16#00,16#00,16#00,16#00,16#00,16#00,16#00,16#00,16#00,16#00,16#00,16#00,	// 16#C1
16#00,16#00,16#00,16#00,16#00,16#00,16#00,16#00,16#00,16#00,16#00,16#00,16#00,16#00,16#00,16#00,16#00,16#00,16#00,16#00,16#00,16#00,16#00,16#00,16#FF,16#FF,16#FF,16#FF,16#80,16#01,16#80,16#01,16#80,16#01,16#80,16#01,16#80,16#01,16#80,16#01,16#80,16#01,16#80,16#01,16#80,16#01,16#80,16#01,16#80,16#01,16#80,16#01,	// 16#C2
16#80,16#01,16#80,16#01,16#80,16#01,16#80,16#01,16#80,16#01,16#80,16#01,16#80,16#01,16#80,16#01,16#80,16#01,16#80,16#01,16#80,16#01,16#80,16#01,16#FF,16#01,16#FF,16#01,16#80,16#01,16#80,16#01,16#80,16#01,16#80,16#01,16#80,16#01,16#80,16#01,16#80,16#01,16#80,16#01,16#80,16#01,16#80,16#01,16#80,16#01,16#80,16#01,	// 16#C3
16#00,16#00,16#00,16#00,16#00,16#00,16#00,16#00,16#00,16#00,16#00,16#00,16#00,16#00,16#00,16#00,16#00,16#00,16#00,16#00,16#00,16#00,16#00,16#00,16#FF,16#FF,16#FF,16#FF,16#00,16#00,16#00,16#00,16#00,16#00,16#00,16#00,16#00,16#00,16#00,16#00,16#00,16#00,16#00,16#00,16#00,16#00,16#00,16#00,16#00,16#00,16#00,16#00,	// 16#C4
16#80,16#01,16#80,16#01,16#80,16#01,16#80,16#01,16#80,16#01,16#80,16#01,16#80,16#01,16#80,16#01,16#80,16#01,16#80,16#01,16#80,16#01,16#80,16#01,16#FF,16#FF,16#FF,16#FF,16#80,16#01,16#80,16#01,16#80,16#01,16#80,16#01,16#80,16#01,16#80,16#01,16#80,16#01,16#80,16#01,16#80,16#01,16#80,16#01,16#80,16#01,16#80,16#01,	// 16#C5
16#00,16#00,16#00,16#00,16#30,16#07,16#F0,16#0F,16#E0,16#0C,16#00,16#00,16#00,16#00,16#E0,16#07,16#F0,16#1F,16#78,16#18,16#38,16#00,16#38,16#00,16#F8,16#07,16#F8,16#0F,16#38,16#1C,16#38,16#38,16#38,16#38,16#38,16#38,16#78,16#3C,16#DE,16#1F,16#1E,16#0F,16#00,16#00,16#00,16#00,16#00,16#00,16#00,16#00,16#00,16#00,	// 16#C6
16#30,16#07,16#F0,16#0F,16#E0,16#0C,16#00,16#00,16#00,16#00,16#80,16#03,16#C0,16#03,16#C0,16#07,16#E0,16#06,16#E0,16#06,16#60,16#0E,16#70,16#0C,16#70,16#1C,16#38,16#1C,16#38,16#18,16#FC,16#3F,16#FC,16#3F,16#1C,16#70,16#0E,16#70,16#0E,16#70,16#07,16#E0,16#00,16#00,16#00,16#00,16#00,16#00,16#00,16#00,16#00,16#00,	// 16#C7
16#60,16#06,16#60,16#06,16#60,16#06,16#60,16#06,16#60,16#06,16#60,16#06,16#60,16#06,16#60,16#06,16#60,16#06,16#60,16#06,16#7F,16#06,16#7F,16#06,16#00,16#06,16#00,16#06,16#FF,16#07,16#FF,16#07,16#00,16#00,16#00,16#00,16#00,16#00,16#00,16#00,16#00,16#00,16#00,16#00,16#00,16#00,16#00,16#00,16#00,16#00,16#00,16#00,	// 16#C8
16#00,16#00,16#00,16#00,16#00,16#00,16#00,16#00,16#00,16#00,16#00,16#00,16#00,16#00,16#00,16#00,16#00,16#00,16#00,16#00,16#FF,16#07,16#FF,16#07,16#00,16#06,16#00,16#06,16#7F,16#06,16#7F,16#06,16#60,16#06,16#60,16#06,16#60,16#06,16#60,16#06,16#60,16#06,16#60,16#06,16#60,16#06,16#60,16#06,16#60,16#06,16#60,16#06,	// 16#C9
16#60,16#06,16#60,16#06,16#60,16#06,16#60,16#06,16#60,16#06,16#60,16#06,16#60,16#06,16#60,16#06,16#60,16#06,16#60,16#06,16#7F,16#FE,16#7F,16#FE,16#00,16#00,16#00,16#00,16#FF,16#FF,16#FF,16#FF,16#00,16#00,16#00,16#00,16#00,16#00,16#00,16#00,16#00,16#00,16#00,16#00,16#00,16#00,16#00,16#00,16#00,16#00,16#00,16#00,	// 16#CA
16#00,16#00,16#00,16#00,16#00,16#00,16#00,16#00,16#00,16#00,16#00,16#00,16#00,16#00,16#00,16#00,16#00,16#00,16#00,16#00,16#FF,16#FF,16#FF,16#FF,16#00,16#00,16#00,16#00,16#7F,16#FE,16#7F,16#FE,16#60,16#06,16#60,16#06,16#60,16#06,16#60,16#06,16#60,16#06,16#60,16#06,16#60,16#06,16#60,16#06,16#60,16#06,16#60,16#06,	// 16#CB
16#60,16#06,16#60,16#06,16#60,16#06,16#60,16#06,16#60,16#06,16#60,16#06,16#60,16#06,16#60,16#06,16#60,16#06,16#60,16#06,16#7F,16#06,16#7F,16#06,16#00,16#06,16#00,16#06,16#7F,16#06,16#7F,16#06,16#60,16#06,16#60,16#06,16#60,16#06,16#60,16#06,16#60,16#06,16#60,16#06,16#60,16#06,16#60,16#06,16#60,16#06,16#60,16#06,	// 16#CC
16#00,16#00,16#00,16#00,16#00,16#00,16#00,16#00,16#00,16#00,16#00,16#00,16#00,16#00,16#00,16#00,16#00,16#00,16#00,16#00,16#FF,16#FF,16#FF,16#FF,16#00,16#00,16#00,16#00,16#FF,16#FF,16#FF,16#FF,16#00,16#00,16#00,16#00,16#00,16#00,16#00,16#00,16#00,16#00,16#00,16#00,16#00,16#00,16#00,16#00,16#00,16#00,16#00,16#00,	// 16#CD
16#60,16#06,16#60,16#06,16#60,16#06,16#60,16#06,16#60,16#06,16#60,16#06,16#60,16#06,16#60,16#06,16#60,16#06,16#60,16#06,16#7F,16#FE,16#7F,16#FE,16#00,16#00,16#00,16#00,16#7F,16#FE,16#7F,16#FE,16#60,16#06,16#60,16#06,16#60,16#06,16#60,16#06,16#60,16#06,16#60,16#06,16#60,16#06,16#60,16#06,16#60,16#06,16#60,16#06,	// 16#CE
16#00,16#00,16#00,16#00,16#00,16#00,16#00,16#00,16#00,16#00,16#00,16#00,16#04,16#20,16#CC,16#33,16#F8,16#1F,16#30,16#0C,16#18,16#18,16#18,16#18,16#18,16#18,16#18,16#18,16#30,16#0C,16#F8,16#1F,16#CC,16#33,16#04,16#20,16#00,16#00,16#00,16#00,16#00,16#00,16#00,16#00,16#00,16#00,16#00,16#00,16#00,16#00,16#00,16#00,	// 16#CF
16#00,16#00,16#C0,16#78,16#C0,16#7F,16#80,16#0F,16#C0,16#0F,16#E0,16#18,16#70,16#00,16#F0,16#07,16#F8,16#1F,16#78,16#3C,16#3C,16#38,16#1C,16#70,16#1C,16#70,16#1C,16#70,16#1C,16#70,16#1C,16#70,16#1C,16#70,16#38,16#38,16#78,16#3C,16#F0,16#1F,16#C0,16#07,16#00,16#00,16#00,16#00,16#00,16#00,16#00,16#00,16#00,16#00,	// 16#D0
16#00,16#00,16#00,16#00,16#00,16#00,16#00,16#00,16#00,16#00,16#E0,16#3F,16#F0,16#3F,16#3C,16#38,16#1C,16#38,16#1E,16#38,16#0E,16#38,16#0E,16#38,16#0E,16#FF,16#0E,16#FF,16#0E,16#38,16#0E,16#38,16#1C,16#38,16#1C,16#38,16#78,16#38,16#F0,16#3F,16#C0,16#3F,16#00,16#00,16#00,16#00,16#00,16#00,16#00,16#00,16#00,16#00,	// 16#D1
16#E0,16#03,16#70,16#07,16#38,16#0E,16#00,16#00,16#00,16#00,16#FC,16#1F,16#FC,16#1F,16#00,16#1C,16#00,16#1C,16#00,16#1C,16#00,16#1C,16#00,16#1C,16#F8,16#1F,16#F8,16#1F,16#00,16#1C,16#00,16#1C,16#00,16#1C,16#00,16#1C,16#00,16#1C,16#FE,16#1F,16#FE,16#1F,16#00,16#00,16#00,16#00,16#00,16#00,16#00,16#00,16#00,16#00,	// 16#D2
16#18,16#06,16#18,16#06,16#00,16#00,16#00,16#00,16#00,16#00,16#FC,16#1F,16#FC,16#1F,16#00,16#1C,16#00,16#1C,16#00,16#1C,16#00,16#1C,16#00,16#1C,16#F8,16#1F,16#F8,16#1F,16#00,16#1C,16#00,16#1C,16#00,16#1C,16#00,16#1C,16#00,16#1C,16#FE,16#1F,16#FE,16#1F,16#00,16#00,16#00,16#00,16#00,16#00,16#00,16#00,16#00,16#00,	// 16#D3
16#80,16#03,16#C0,16#01,16#E0,16#00,16#00,16#00,16#00,16#00,16#FC,16#1F,16#FC,16#1F,16#00,16#1C,16#00,16#1C,16#00,16#1C,16#00,16#1C,16#00,16#1C,16#F8,16#1F,16#F8,16#1F,16#00,16#1C,16#00,16#1C,16#00,16#1C,16#00,16#1C,16#00,16#1C,16#FE,16#1F,16#FE,16#1F,16#00,16#00,16#00,16#00,16#00,16#00,16#00,16#00,16#00,16#00,	// 16#D4
16#00,16#00,16#00,16#00,16#00,16#00,16#00,16#00,16#00,16#00,16#00,16#00,16#00,16#00,16#C0,16#3F,16#C0,16#3F,16#C0,16#01,16#C0,16#01,16#C0,16#01,16#C0,16#01,16#C0,16#01,16#C0,16#01,16#C0,16#01,16#C0,16#01,16#C0,16#01,16#C0,16#01,16#C0,16#01,16#C0,16#01,16#00,16#00,16#00,16#00,16#00,16#00,16#00,16#00,16#00,16#00,	// 16#D5
16#E0,16#00,16#C0,16#01,16#80,16#03,16#00,16#00,16#00,16#00,16#F8,16#3F,16#F8,16#3F,16#80,16#03,16#80,16#03,16#80,16#03,16#80,16#03,16#80,16#03,16#80,16#03,16#80,16#03,16#80,16#03,16#80,16#03,16#80,16#03,16#80,16#03,16#80,16#03,16#F8,16#3F,16#F8,16#3F,16#00,16#00,16#00,16#00,16#00,16#00,16#00,16#00,16#00,16#00,	// 16#D6
16#C0,16#07,16#E0,16#0E,16#70,16#1C,16#00,16#00,16#00,16#00,16#F8,16#3F,16#F8,16#3F,16#80,16#03,16#80,16#03,16#80,16#03,16#80,16#03,16#80,16#03,16#80,16#03,16#80,16#03,16#80,16#03,16#80,16#03,16#80,16#03,16#80,16#03,16#80,16#03,16#F8,16#3F,16#F8,16#3F,16#00,16#00,16#00,16#00,16#00,16#00,16#00,16#00,16#00,16#00,	// 16#D7
16#30,16#0C,16#30,16#0C,16#00,16#00,16#00,16#00,16#00,16#00,16#F8,16#3F,16#F8,16#3F,16#80,16#03,16#80,16#03,16#80,16#03,16#80,16#03,16#80,16#03,16#80,16#03,16#80,16#03,16#80,16#03,16#80,16#03,16#80,16#03,16#80,16#03,16#80,16#03,16#F8,16#3F,16#F8,16#3F,16#00,16#00,16#00,16#00,16#00,16#00,16#00,16#00,16#00,16#00,	// 16#D8
16#80,16#01,16#80,16#01,16#80,16#01,16#80,16#01,16#80,16#01,16#80,16#01,16#80,16#01,16#80,16#01,16#80,16#01,16#80,16#01,16#80,16#01,16#80,16#01,16#80,16#FF,16#80,16#FF,16#00,16#00,16#00,16#00,16#00,16#00,16#00,16#00,16#00,16#00,16#00,16#00,16#00,16#00,16#00,16#00,16#00,16#00,16#00,16#00,16#00,16#00,16#00,16#00,	// 16#D9
16#00,16#00,16#00,16#00,16#00,16#00,16#00,16#00,16#00,16#00,16#00,16#00,16#00,16#00,16#00,16#00,16#00,16#00,16#00,16#00,16#00,16#00,16#00,16#00,16#FF,16#01,16#FF,16#01,16#80,16#01,16#80,16#01,16#80,16#01,16#80,16#01,16#80,16#01,16#80,16#01,16#80,16#01,16#80,16#01,16#80,16#01,16#80,16#01,16#80,16#01,16#80,16#01,	// 16#DA
16#FF,16#FF,16#FF,16#FF,16#FF,16#FF,16#FF,16#FF,16#FF,16#FF,16#FF,16#FF,16#FF,16#FF,16#FF,16#FF,16#FF,16#FF,16#FF,16#FF,16#FF,16#FF,16#FF,16#FF,16#FF,16#FF,16#FF,16#FF,16#FF,16#FF,16#FF,16#FF,16#FF,16#FF,16#FF,16#FF,16#FF,16#FF,16#FF,16#FF,16#FF,16#FF,16#FF,16#FF,16#FF,16#FF,16#FF,16#FF,16#FF,16#FF,16#FF,16#FF,	// 16#DB
16#00,16#00,16#00,16#00,16#00,16#00,16#00,16#00,16#00,16#00,16#00,16#00,16#00,16#00,16#00,16#00,16#00,16#00,16#00,16#00,16#00,16#00,16#00,16#00,16#00,16#00,16#FF,16#FF,16#FF,16#FF,16#FF,16#FF,16#FF,16#FF,16#FF,16#FF,16#FF,16#FF,16#FF,16#FF,16#FF,16#FF,16#FF,16#FF,16#FF,16#FF,16#FF,16#FF,16#FF,16#FF,16#FF,16#FF,	// 16#DC
16#00,16#00,16#80,16#01,16#80,16#01,16#80,16#01,16#80,16#01,16#80,16#01,16#80,16#01,16#80,16#01,16#80,16#01,16#80,16#01,16#00,16#00,16#00,16#00,16#00,16#00,16#00,16#00,16#00,16#00,16#80,16#01,16#80,16#01,16#80,16#01,16#80,16#01,16#80,16#01,16#80,16#01,16#80,16#01,16#80,16#01,16#80,16#01,16#80,16#01,16#00,16#00,	// 16#DD
16#00,16#07,16#80,16#03,16#C0,16#01,16#00,16#00,16#00,16#00,16#F8,16#3F,16#F8,16#3F,16#80,16#03,16#80,16#03,16#80,16#03,16#80,16#03,16#80,16#03,16#80,16#03,16#80,16#03,16#80,16#03,16#80,16#03,16#80,16#03,16#80,16#03,16#80,16#03,16#F8,16#3F,16#F8,16#3F,16#00,16#00,16#00,16#00,16#00,16#00,16#00,16#00,16#00,16#00,	// 16#DE
16#FF,16#FF,16#FF,16#FF,16#FF,16#FF,16#FF,16#FF,16#FF,16#FF,16#FF,16#FF,16#FF,16#FF,16#FF,16#FF,16#FF,16#FF,16#FF,16#FF,16#FF,16#FF,16#FF,16#FF,16#FF,16#FF,16#00,16#00,16#00,16#00,16#00,16#00,16#00,16#00,16#00,16#00,16#00,16#00,16#00,16#00,16#00,16#00,16#00,16#00,16#00,16#00,16#00,16#00,16#00,16#00,16#00,16#00,	// 16#DF
16#E0,16#00,16#C0,16#01,16#80,16#03,16#00,16#00,16#00,16#00,16#E0,16#07,16#F0,16#0F,16#38,16#1C,16#1C,16#38,16#1C,16#38,16#0E,16#70,16#0E,16#70,16#0E,16#70,16#0E,16#70,16#0E,16#70,16#0E,16#70,16#1C,16#38,16#1C,16#38,16#38,16#1C,16#F0,16#0F,16#E0,16#07,16#00,16#00,16#00,16#00,16#00,16#00,16#00,16#00,16#00,16#00,	// 16#E0
16#00,16#00,16#C0,16#0F,16#E0,16#1F,16#70,16#3C,16#70,16#38,16#70,16#38,16#60,16#38,16#E0,16#38,16#C0,16#39,16#C0,16#39,16#C0,16#39,16#E0,16#39,16#F0,16#38,16#78,16#38,16#3C,16#38,16#1E,16#38,16#0E,16#38,16#0E,16#38,16#0E,16#39,16#FC,16#39,16#F8,16#38,16#00,16#00,16#00,16#00,16#00,16#00,16#00,16#00,16#00,16#00,	// 16#E1
16#C0,16#07,16#E0,16#0E,16#70,16#1C,16#00,16#00,16#00,16#00,16#E0,16#07,16#F0,16#0F,16#38,16#1C,16#1C,16#38,16#1C,16#38,16#0E,16#70,16#0E,16#70,16#0E,16#70,16#0E,16#70,16#0E,16#70,16#0E,16#70,16#1C,16#38,16#1C,16#38,16#38,16#1C,16#F0,16#0F,16#E0,16#07,16#00,16#00,16#00,16#00,16#00,16#00,16#00,16#00,16#00,16#00,	// 16#E2
16#00,16#07,16#80,16#03,16#C0,16#01,16#00,16#00,16#00,16#00,16#E0,16#07,16#F0,16#0F,16#38,16#1C,16#1C,16#38,16#1C,16#38,16#0E,16#70,16#0E,16#70,16#0E,16#70,16#0E,16#70,16#0E,16#70,16#0E,16#70,16#1C,16#38,16#1C,16#38,16#38,16#1C,16#F0,16#0F,16#E0,16#07,16#00,16#00,16#00,16#00,16#00,16#00,16#00,16#00,16#00,16#00,	// 16#E3
16#00,16#00,16#00,16#00,16#30,16#07,16#F0,16#0F,16#E0,16#0C,16#00,16#00,16#00,16#00,16#C0,16#07,16#F0,16#1F,16#78,16#3C,16#38,16#38,16#1C,16#70,16#1C,16#70,16#1C,16#70,16#1C,16#70,16#1C,16#70,16#1C,16#70,16#38,16#38,16#78,16#3C,16#F0,16#1F,16#C0,16#07,16#00,16#00,16#00,16#00,16#00,16#00,16#00,16#00,16#00,16#00,	// 16#E4
16#30,16#07,16#F0,16#0F,16#E0,16#0C,16#00,16#00,16#00,16#00,16#E0,16#07,16#F0,16#0F,16#38,16#1C,16#1C,16#38,16#1C,16#38,16#0E,16#70,16#0E,16#70,16#0E,16#70,16#0E,16#70,16#0E,16#70,16#0E,16#70,16#1C,16#38,16#1C,16#38,16#38,16#1C,16#F0,16#0F,16#E0,16#07,16#00,16#00,16#00,16#00,16#00,16#00,16#00,16#00,16#00,16#00,	// 16#E5
16#00,16#00,16#00,16#00,16#00,16#00,16#00,16#00,16#00,16#00,16#00,16#00,16#00,16#00,16#1C,16#38,16#1C,16#38,16#1C,16#38,16#1C,16#38,16#1C,16#38,16#1C,16#38,16#1C,16#38,16#1C,16#38,16#1C,16#38,16#1C,16#38,16#3C,16#3C,16#7C,16#3E,16#DC,16#3F,16#DE,16#3B,16#00,16#38,16#00,16#38,16#00,16#38,16#00,16#38,16#00,16#38,	// 16#E6
16#00,16#00,16#00,16#38,16#00,16#38,16#00,16#38,16#00,16#38,16#00,16#38,16#00,16#38,16#E0,16#39,16#F8,16#3B,16#38,16#3E,16#1C,16#3C,16#1C,16#38,16#1C,16#38,16#1C,16#38,16#1C,16#38,16#1C,16#38,16#1C,16#38,16#38,16#38,16#78,16#3C,16#F0,16#3F,16#E0,16#39,16#00,16#38,16#00,16#38,16#00,16#38,16#00,16#38,16#00,16#38,	// 16#E7
16#00,16#00,16#00,16#00,16#00,16#00,16#00,16#00,16#00,16#00,16#00,16#1C,16#00,16#1C,16#00,16#1C,16#F8,16#1F,16#FC,16#1F,16#1E,16#1C,16#0E,16#1C,16#0E,16#1C,16#0E,16#1C,16#1E,16#1C,16#3C,16#1C,16#F8,16#1F,16#E0,16#1F,16#00,16#1C,16#00,16#1C,16#00,16#1C,16#00,16#00,16#00,16#00,16#00,16#00,16#00,16#00,16#00,16#00,	// 16#E8
16#E0,16#00,16#C0,16#01,16#80,16#03,16#00,16#00,16#00,16#00,16#0E,16#38,16#0E,16#38,16#0E,16#38,16#0E,16#38,16#0E,16#38,16#0E,16#38,16#0E,16#38,16#0E,16#38,16#0E,16#38,16#0E,16#38,16#0E,16#38,16#0E,16#38,16#1E,16#3C,16#1C,16#1C,16#F8,16#0F,16#F0,16#07,16#00,16#00,16#00,16#00,16#00,16#00,16#00,16#00,16#00,16#00,	// 16#E9
16#C0,16#07,16#E0,16#0E,16#70,16#1C,16#00,16#00,16#00,16#00,16#0E,16#38,16#0E,16#38,16#0E,16#38,16#0E,16#38,16#0E,16#38,16#0E,16#38,16#0E,16#38,16#0E,16#38,16#0E,16#38,16#0E,16#38,16#0E,16#38,16#0E,16#38,16#1E,16#3C,16#1C,16#1C,16#F8,16#0F,16#F0,16#07,16#00,16#00,16#00,16#00,16#00,16#00,16#00,16#00,16#00,16#00,	// 16#EA
16#00,16#07,16#80,16#03,16#C0,16#01,16#00,16#00,16#00,16#00,16#0E,16#38,16#0E,16#38,16#0E,16#38,16#0E,16#38,16#0E,16#38,16#0E,16#38,16#0E,16#38,16#0E,16#38,16#0E,16#38,16#0E,16#38,16#0E,16#38,16#0E,16#38,16#1E,16#3C,16#1C,16#1C,16#F8,16#0F,16#F0,16#07,16#00,16#00,16#00,16#00,16#00,16#00,16#00,16#00,16#00,16#00,	// 16#EB
16#00,16#00,16#60,16#00,16#C0,16#00,16#80,16#01,16#00,16#03,16#00,16#00,16#00,16#00,16#0E,16#78,16#0C,16#38,16#1C,16#38,16#18,16#1C,16#38,16#1C,16#38,16#1E,16#70,16#0E,16#70,16#0F,16#E0,16#07,16#E0,16#07,16#C0,16#03,16#C0,16#03,16#80,16#03,16#80,16#01,16#80,16#03,16#00,16#03,16#00,16#07,16#00,16#3E,16#00,16#3C,	// 16#EC
16#E0,16#00,16#C0,16#01,16#80,16#03,16#00,16#00,16#00,16#00,16#07,16#E0,16#0E,16#70,16#0C,16#38,16#18,16#38,16#38,16#1C,16#70,16#1E,16#E0,16#0E,16#C0,16#07,16#C0,16#07,16#80,16#03,16#80,16#03,16#80,16#03,16#80,16#03,16#80,16#03,16#80,16#03,16#80,16#03,16#00,16#00,16#00,16#00,16#00,16#00,16#00,16#00,16#00,16#00,	// 16#ED
16#FF,16#FF,16#FF,16#FF,16#00,16#00,16#00,16#00,16#00,16#00,16#00,16#00,16#00,16#00,16#00,16#00,16#00,16#00,16#00,16#00,16#00,16#00,16#00,16#00,16#00,16#00,16#00,16#00,16#00,16#00,16#00,16#00,16#00,16#00,16#00,16#00,16#00,16#00,16#00,16#00,16#00,16#00,16#00,16#00,16#00,16#00,16#00,16#00,16#00,16#00,16#00,16#00,	// 16#EE
16#C0,16#01,16#80,16#03,16#00,16#07,16#00,16#00,16#00,16#00,16#00,16#00,16#00,16#00,16#00,16#00,16#00,16#00,16#00,16#00,16#00,16#00,16#00,16#00,16#00,16#00,16#00,16#00,16#00,16#00,16#00,16#00,16#00,16#00,16#00,16#00,16#00,16#00,16#00,16#00,16#00,16#00,16#00,16#00,16#00,16#00,16#00,16#00,16#00,16#00,16#00,16#00,	// 16#EF
16#00,16#00,16#00,16#00,16#00,16#00,16#00,16#00,16#00,16#00,16#00,16#00,16#00,16#00,16#00,16#00,16#00,16#00,16#00,16#00,16#00,16#00,16#00,16#00,16#F8,16#1F,16#F8,16#1F,16#00,16#00,16#00,16#00,16#00,16#00,16#00,16#00,16#00,16#00,16#00,16#00,16#00,16#00,16#00,16#00,16#00,16#00,16#00,16#00,16#00,16#00,16#00,16#00,	// 16#F0
16#00,16#00,16#00,16#00,16#00,16#00,16#00,16#00,16#00,16#00,16#00,16#00,16#00,16#00,16#80,16#01,16#80,16#01,16#80,16#01,16#80,16#01,16#FE,16#7F,16#FE,16#7F,16#80,16#01,16#80,16#01,16#80,16#01,16#80,16#01,16#00,16#00,16#00,16#00,16#FE,16#7F,16#FE,16#7F,16#00,16#00,16#00,16#00,16#00,16#00,16#00,16#00,16#00,16#00,	// 16#F1
16#00,16#00,16#00,16#00,16#00,16#00,16#00,16#00,16#00,16#00,16#00,16#00,16#00,16#00,16#00,16#00,16#00,16#00,16#00,16#00,16#00,16#00,16#00,16#00,16#00,16#00,16#00,16#00,16#00,16#00,16#00,16#00,16#00,16#00,16#00,16#00,16#00,16#00,16#00,16#00,16#00,16#00,16#FF,16#FF,16#FF,16#FF,16#00,16#00,16#00,16#00,16#FF,16#FF,	// 16#F2
16#00,16#00,16#00,16#00,16#07,16#7E,16#0E,16#7F,16#1C,16#07,16#1C,16#07,16#38,16#3C,16#38,16#3E,16#70,16#07,16#E0,16#07,16#E0,16#7F,16#DC,16#7D,16#BC,16#03,16#DC,16#03,16#9C,16#07,16#9C,16#0F,16#1C,16#0F,16#FF,16#1F,16#1C,16#1C,16#1C,16#38,16#1C,16#70,16#00,16#00,16#00,16#00,16#00,16#00,16#00,16#00,16#00,16#00,	// 16#F3
16#00,16#00,16#00,16#00,16#F8,16#1F,16#F8,16#3F,16#18,16#7F,16#18,16#7F,16#18,16#7F,16#18,16#7F,16#18,16#7F,16#18,16#3F,16#18,16#1F,16#18,16#0F,16#18,16#03,16#18,16#03,16#18,16#03,16#18,16#03,16#18,16#03,16#18,16#03,16#18,16#03,16#18,16#03,16#18,16#03,16#18,16#03,16#18,16#03,16#18,16#03,16#18,16#03,16#00,16#00,	// 16#F4
16#00,16#00,16#00,16#00,16#F8,16#03,16#F8,16#0F,16#08,16#1E,16#00,16#1C,16#00,16#1C,16#00,16#1E,16#80,16#0F,16#E0,16#07,16#F0,16#0F,16#78,16#0C,16#3C,16#1C,16#1C,16#1C,16#1C,16#1E,16#98,16#0F,16#F0,16#07,16#F0,16#01,16#78,16#00,16#3C,16#00,16#1C,16#00,16#1C,16#00,16#3C,16#18,16#F8,16#1F,16#E0,16#07,16#00,16#00,	// 16#F5
16#00,16#00,16#00,16#00,16#00,16#00,16#00,16#00,16#00,16#00,16#00,16#00,16#00,16#00,16#80,16#03,16#80,16#03,16#80,16#03,16#00,16#00,16#00,16#00,16#00,16#00,16#FC,16#7F,16#FC,16#7F,16#00,16#00,16#00,16#00,16#00,16#00,16#80,16#03,16#80,16#03,16#80,16#03,16#00,16#00,16#00,16#00,16#00,16#00,16#00,16#00,16#00,16#00,	// 16#F6
16#00,16#00,16#00,16#00,16#00,16#00,16#00,16#00,16#00,16#00,16#00,16#00,16#00,16#00,16#00,16#00,16#00,16#00,16#00,16#00,16#00,16#00,16#00,16#00,16#00,16#00,16#00,16#00,16#00,16#00,16#00,16#00,16#00,16#00,16#00,16#00,16#00,16#00,16#00,16#00,16#00,16#00,16#80,16#00,16#C0,16#01,16#60,16#00,16#60,16#00,16#C0,16#03,	// 16#F7
16#00,16#00,16#00,16#00,16#00,16#07,16#80,16#08,16#80,16#08,16#80,16#08,16#00,16#07,16#00,16#00,16#00,16#00,16#00,16#00,16#00,16#00,16#00,16#00,16#00,16#00,16#00,16#00,16#00,16#00,16#00,16#00,16#00,16#00,16#00,16#00,16#00,16#00,16#00,16#00,16#00,16#00,16#00,16#00,16#00,16#00,16#00,16#00,16#00,16#00,16#00,16#00,	// 16#F8
16#30,16#0C,16#30,16#0C,16#00,16#00,16#00,16#00,16#00,16#00,16#00,16#00,16#00,16#00,16#00,16#00,16#00,16#00,16#00,16#00,16#00,16#00,16#00,16#00,16#00,16#00,16#00,16#00,16#00,16#00,16#00,16#00,16#00,16#00,16#00,16#00,16#00,16#00,16#00,16#00,16#00,16#00,16#00,16#00,16#00,16#00,16#00,16#00,16#00,16#00,16#00,16#00,	// 16#F9
16#00,16#00,16#00,16#00,16#00,16#00,16#00,16#00,16#00,16#00,16#00,16#00,16#00,16#00,16#00,16#00,16#00,16#00,16#00,16#00,16#00,16#00,16#00,16#00,16#00,16#00,16#80,16#03,16#80,16#03,16#80,16#03,16#00,16#00,16#00,16#00,16#00,16#00,16#00,16#00,16#00,16#00,16#00,16#00,16#00,16#00,16#00,16#00,16#00,16#00,16#00,16#00,	// 16#FA
16#00,16#00,16#00,16#00,16#C0,16#07,16#C0,16#07,16#C0,16#01,16#C0,16#01,16#C0,16#01,16#C0,16#01,16#C0,16#01,16#C0,16#01,16#C0,16#01,16#C0,16#01,16#00,16#00,16#00,16#00,16#00,16#00,16#00,16#00,16#00,16#00,16#00,16#00,16#00,16#00,16#00,16#00,16#00,16#00,16#00,16#00,16#00,16#00,16#00,16#00,16#00,16#00,16#00,16#00,	// 16#FB
16#00,16#00,16#00,16#00,16#F0,16#07,16#F8,16#0F,16#38,16#08,16#38,16#00,16#E0,16#03,16#F0,16#03,16#38,16#00,16#38,16#00,16#F8,16#0F,16#E0,16#0F,16#00,16#00,16#00,16#00,16#00,16#00,16#00,16#00,16#00,16#00,16#00,16#00,16#00,16#00,16#00,16#00,16#00,16#00,16#00,16#00,16#00,16#00,16#00,16#00,16#00,16#00,16#00,16#00,	// 16#FC
16#00,16#00,16#00,16#00,16#E0,16#07,16#F8,16#0F,16#38,16#08,16#38,16#00,16#70,16#00,16#E0,16#01,16#80,16#03,16#00,16#0E,16#F8,16#0F,16#F8,16#0F,16#00,16#00,16#00,16#00,16#00,16#00,16#00,16#00,16#00,16#00,16#00,16#00,16#00,16#00,16#00,16#00,16#00,16#00,16#00,16#00,16#00,16#00,16#00,16#00,16#00,16#00,16#00,16#00,	// 16#FD
16#00,16#00,16#00,16#00,16#00,16#00,16#00,16#00,16#00,16#00,16#00,16#00,16#00,16#00,16#FE,16#7F,16#FE,16#7F,16#FE,16#7F,16#FE,16#7F,16#FE,16#7F,16#FE,16#7F,16#FE,16#7F,16#FE,16#7F,16#FE,16#7F,16#FE,16#7F,16#FE,16#7F,16#FE,16#7F,16#FE,16#7F,16#FE,16#7F,16#00,16#00,16#00,16#00,16#00,16#00,16#00,16#00,16#00,16#00,	// 16#FE
16#00,16#00,16#00,16#00,16#00,16#00,16#00,16#00,16#00,16#00,16#00,16#00,16#00,16#00,16#00,16#00,16#00,16#00,16#00,16#00,16#00,16#00,16#00,16#00,16#00,16#00,16#00,16#00,16#00,16#00,16#00,16#00,16#00,16#00,16#00,16#00,16#00,16#00,16#00,16#00,16#00,16#00,16#00,16#00,16#00,16#00,16#00,16#00,16#00,16#00,16#00,16#00 	// 16#FF
];


END_VAR

SUPER^();

METHOD Initialize : UDINT
VAR_INPUT
	wModuleType : UINT;
	dwInstance : UDINT;
	pConnector : POINTER TO IoConfigConnector;
END_VAR
VAR
	pParam: POINTER TO IoConfigParameter;		
	udiResult: UDINT;
	byte1:BYTE;
	i:int;	
END_VAR
SUPER^.Initialize(wModuleType, dwInstance, pConnector);

pParam := ConfigGetParameter(_pConnector, 20);
displayHeight:= IoStandard.ConfigGetParameterValueByte(pParam, ADR(udiResult));

pParam := ConfigGetParameter(_pConnector, 21);
displayWidth:= IoStandard.ConfigGetParameterValueByte(pParam, ADR(udiResult));

displaySize := displayHeight * displayWidth;


bytesPerRow := displayWidth;

stateAfterError := START_DEVICE;
stateAfterInit := START_DEVICE;
(*
FOR i := 0 TO SIZEOF(displayBuffer)-1 DO
	displayBuffer[i+1]:=bitmask[i MOD 8];
END_FOR
*)
END_METHOD

METHOD BeforeWriteOutputs : INT
VAR
	


END_VAR
SUPER^.BeforeWriteOutputs();
IF NOT UseEnableWire THEN
	IF checkInitMultiplex() THEN
		RETURN;
	END_IF
ELSE
	IF NOT enableInstanceSet THEN
		RETURN;
	END_IF
END_IF
//GVL.callNum := 0;
IF checkInitMultiplex() THEN
	RETURN;
END_IF
CASE _iState OF
START_DEVICE:
	writeRequest.request := TRUE;
	IF NOT (setWire() = SET_SLAVE_NUM_RETURN.NUM_IO) AND UseEnableWire THEN
		RETURN;
	END_IF
	IF NOT checkWriteTimeMultiplex(ADR(writeRequest)) THEN
		RETURN;
	END_IF 
	writeRequestLCDData := FALSE;
	//write init data
	//16#A8, 63,		// Set multiplex ratio(1 to 64)
	initDisplayData[SIZEOF(initDisplayData)-2]:=16#A8;
	initDisplayData[SIZEOF(initDisplayData)-1]:=displayHeight - 1;
	checkWrite(pbyBuffer:= ADR(initDisplayData), nBufferLen:= SIZEOF(initDisplayData));

	IF _iState<>ERROR_DEVICE THEN
		_iState := RUN_DEVICE;	 
	END_IF
	releaseWire();

RUN_DEVICE:
	//requestWrite
	IF writeRequestLCDData OR writeRequestLCDCommand THEN
		writeRequest.request := TRUE;
	ELSE
		RETURN;
	END_IF
	IF NOT (setWire() = SET_SLAVE_NUM_RETURN.NUM_IO) AND UseEnableWire THEN
		RETURN;
	END_IF
	IF NOT checkWriteTimeMultiplex(ADR(writeRequest)) THEN
		RETURN;
	END_IF
	//reset request
	writeRequest.request := FALSE;
	IF writeRequestLCDData THEN
		lastBufferWriteTime := TICKS.GetTick(xDummy:= TRUE);
		checkWrite(pbyBuffer:= ADR(displayBuffer), nBufferLen:= SIZEOF(displayBuffer));
		lastBufferWriteTime := TICKS.GetTick(xDummy:= TRUE) - lastBufferWriteTime;
		writeRequestLCDData := FALSE;
	END_IF
	
	IF writeRequestLCDCommand THEN
		checkWrite(pbyBuffer:= ADR(commandBuffer), nBufferLen:= sizeOfCommands);
		sizeOfCommands := 1;
		writeRequestLCDCommand := FALSE;
	END_IF
	releaseWire();
	
END_CASE
END_METHOD

METHOD DisplayOn
VAR_INPUT
END_VAR
VAR CONSTANT
	command:ARRAY[0..0]OF BYTE := [16#AF];
END_VAR
displayOnOff := TRUE;

writeRequestLCDCommand := TRUE;

SetCommand(command := command);
END_METHOD

METHOD DisplayOff
VAR_INPUT
END_VAR
VAR CONSTANT
	command:ARRAY[0..0]OF BYTE := [16#AE];
END_VAR
displayOnOff := FALSE;

writeRequestLCDCommand := TRUE;

SetCommand(command := command);
END_METHOD

METHOD SetCommand
VAR_IN_OUT
	command:ARRAY[*] OF BYTE;	
END_VAR

VAR_INPUT 


END_VAR
VAR
	i: DINT;
END_VAR

writeRequestLCDCommand := TRUE;

FOR i := LOWER_BOUND(command, 1) TO UPPER_BOUND(command, 1) DO
	commandBuffer[sizeOfCommands] := command[i];
	sizeOfCommands := sizeOfCommands + 1;
	
END_FOR
END_METHOD

METHOD SetContrast
VAR_INPUT
	contrast:BYTE;
	
END_VAR
VAR
	command:ARRAY[0..1]OF BYTE :=[16#81];
	
END_VAR
command[1]:=contrast;

SetCommand(command:= command);
END_METHOD

METHOD DrawLine
VAR_INPUT
	x1:USINT;
	y1:USINT;
	x2:USINT;
	y2:USINT;
	mode:USINT;
END_VAR
VAR
	dy:INT;
	dx:INT;
	stepx:INT;
	stepy:INT;
	fraction:INT;
	mask:BYTE;
	i:INT;
	address: POINTER TO BYTE;
	countBytes :USINT;
	yStart:BYTE;
	yEnd:BYTE;
END_VAR
IF y1 = y2 THEN
	IF x2 < x1 THEN
		//swap x1 and x2
		mask := x1;
		x1 := x2;
		x2 := mask;
	END_IF
	mask := bitMask[x1 MOD 8];
	//no go over the bits
	address := ADR(displayBuffer)+(y1 / PixPerByte) * BytesPerRow;
	address := address + (x1 MOD BytesPerRow);
	address := address + 1;//one Byte for command identifier
	CASE mode OF
		LCD_MODES.CLEAR_BIT:
			//invert mask for clearing
			mask := NOT mask;
			FOR i := 0 TO x2 - x1 DO
				address^ := address^ AND mask;	
				address := address + 1;
			END_FOR
		LCD_MODES.SET_BIT:
			FOR i := 0 TO x2 - x1 DO
				address^ := address^ OR mask;	
				address := address + 1;
			END_FOR
		LCD_MODES.INVERT_BIT:
			FOR i := 0 TO x2 - x1 DO
				address^ := address^ XOR mask;	
				address := address + 1;
			END_FOR 
	END_CASE
	RETURN;
END_IF

IF x1 = x2 AND 0 THEN
	IF y2 < y1 THEN
		mask := y1;
		y1 := y2;
		y2 := mask;
		address := ADR(displayBuffer)+(y1 / PixPerByte) * BytesPerRow;
		address := address + (x1 MOD BytesPerRow);
		address := address + 1;//one Byte for command identifier	
		yStart := byteMask[(y1 MOD 8) + 8];
		yEnd := byteMask[(y2 MOD 8)];
		countBytes := y1 / 8 - y2 / 8;
		IF countBytes = 0 THEN
			//just one byte to handle
			CASE mode OF
			LCD_MODES.CLEAR_BIT:
				//invert mask for clearing
				mask := NOT (yStart OR yEnd);
				address^ := address^ AND mask;	
			LCD_MODES.SET_BIT:
				address^ := address^ OR (yStart OR yEnd);	
			LCD_MODES.INVERT_BIT:
				address^ := address^ XOR (yStart OR yEnd);
			END_CASE		
			RETURN;
		END_IF
		//more then one byte here
		CASE mode OF
			LCD_MODES.CLEAR_BIT:
				address^ := address^ AND NOT yStart;
				address := address + BytesPerRow;
				WHILE countBytes <> 0 DO
					address^ := 0;	
					address := address + BytesPerRow;
				END_WHILE
				address^ := address^ AND NOT yEnd;
			LCD_MODES.SET_BIT:
				address^ := address^ OR yStart;
				address := address + BytesPerRow;
				WHILE countBytes <> 0 DO
					address^ := 16#FF;	
					address := address + BytesPerRow;
				END_WHILE
				address^ := address^ OR yEnd;
			LCD_MODES.INVERT_BIT:
				address^ := address^ XOR yStart;
				address := address + BytesPerRow;
				WHILE countBytes <> 0 DO
					address^ := address^ XOR 16#FF;	
					address := address + BytesPerRow;
				END_WHILE
				address^ := address^ XOR yEnd; 
		END_CASE		
			
	END_IF
	RETURN;
END_IF

dy := y2 - y1;
dx := x2 - x1;
	IF (dy < 0) THEN
		dy := -dy;
		stepy := -1;
	 ELSE 
		stepy := 1;
	END_IF
	IF (dx < 0) THEN
		dx := -dx;
		stepx := -1;
	 ELSE 
		stepx := 1;
	END_IF
	dy :=SHL(dy,1);
	dx :=SHL(dx,1);
	
	SetPixelCache(xPos:= x1, yPos:= y1, mode:= mode);
IF (dx > dy) THEN
	fraction := dy - SHR(dx, 1);
	WHILE (x1 <> x2) DO
		IF (fraction >= 0) THEN
			y1 := INT_TO_USINT(y1 + stepy);
			fraction := fraction - dx; 
		END_IF
		x1 := INT_TO_USINT(x1 + stepx);
		fraction := fraction + dy;
		SetPixelCache(xPos:= x1, yPos:= y1, mode:= mode);
	END_WHILE
 ELSE 
	fraction := dx - SHR(dy, 1);
	WHILE (y1 <> y2) DO
		IF (fraction >= 0) THEN
			x1 := INT_TO_USINT(x1 + stepx);
			fraction := fraction - dy;
		END_IF
		y1 := INT_TO_USINT(y1 + stepy);
		fraction := fraction + dx;
		SetPixelCache(xPos:= x1, yPos:= y1, mode:= mode);
	END_WHILE
END_IF
END_METHOD

METHOD SetPixelCache
VAR_INPUT
	xPos:USINT;
	yPos:USINT;
	mode:USINT;
END_VAR
VAR
	address:UINT;
	mask:BYTE;
	cacheByte:byte;
END_VAR
// Byte im LCD Cach aussrechnen
//calculoate byte in cache
IF xpos >= displayWidth OR ypos >= displayHeight THEN RETURN; END_IF
address := (ypos / PixPerByte) * BytesPerRow;
address := address + (xpos MOD BytesPerRow);
mask := bitMask[ypos MOD pixPerByte];
cacheByte := GetCacheByte(address:= address);
CASE mode OF
	LCD_MODES.SET_BIT:
		cacheByte := cacheByte OR mask;
	LCD_MODES.CLEAR_BIT:
		cacheByte := cacheByte AND NOT mask;
	LCD_MODES.INVERT_BIT:
		cacheByte := cacheByte XOR mask;
END_CASE

SetCacheByteRaw(address:= address, cacheByte:= cacheByte);
END_METHOD

METHOD GetCacheByte : byte
VAR_INPUT
	address:UINT;
END_VAR
GetCacheByte := displayBuffer[address + 1];
END_METHOD

METHOD SetCacheByteRaw
VAR_INPUT
	address:UINT;
	cacheByte:byte;
END_VAR
displayBuffer[address + 1] := cacheByte;
END_METHOD

METHOD WriteCacheToLcd
VAR_INPUT
END_VAR
writeRequestLCDData := true;
END_METHOD

METHOD SetByteCache
VAR_INPUT
	xpos:USINT;
	ypos:USINT;
	data:USINT;
	mask:USINT;
	mode:USINT;
	
END_VAR
VAR
	address:UINT;
	tmpMask:WORD;
	tmpData:WORD;
	byteDisplacement:USINT;
	cacheByte1: BYTE;
	cacheByte2: BYTE;
END_VAR
IF xpos >= displayWidth OR ypos >= displayHeight THEN RETURN; END_IF

address := (ypos / PixPerByte) * BytesPerRow;
address := address + (xpos MOD BytesPerRow);
byteDisplacement := ypos MOD pixPerByte;
cacheByte1 := GetCacheByte(address:= address);

IF byteDisplacement = 0 THEN
	//one byte opperation
	CASE mode OF
		LCD_MODES.CLEAR_BIT:
			cacheByte1 := cacheByte1 AND NOT data;
		LCD_MODES.SET_BIT:
			cacheByte1 := cacheByte1 AND NOT mask;
			cacheByte1 := cacheByte1 OR data;
		LCD_MODES.INVERT_BIT:
			cacheByte1 := cacheByte1 XOR data;
	END_CASE
	SetCacheByteRaw(address:= address, cacheByte:= cacheByte1);
ELSE
	//two byte opperation
	(*tmpMask := SHL(mask, 8 - byteDisplacement);
	tmpData := SHL(data, 8 - byteDisplacement);*)
	tmpMask := SHL(BYTE_TO_WORD(mask), byteDisplacement);
	tmpData := SHL(BYTE_TO_WORD(data), byteDisplacement);
	IF ypos > displayHeight - 8 THEN
		//second byte is out of display
		CASE mode OF
			LCD_MODES.CLEAR_BIT:
				cacheByte1 := WORD_TO_BYTE(cacheByte1 AND NOT tmpData);
			LCD_MODES.SET_BIT:
				cacheByte1 := WORD_TO_BYTE(cacheByte1 AND NOT tmpMask);
				cacheByte1 := WORD_TO_BYTE(cacheByte1 OR tmpData);
			LCD_MODES.INVERT_BIT:
				cacheByte1 := WORD_TO_BYTE(cacheByte1 XOR tmpData);
		END_CASE
		SetCacheByteRaw(address:= address, cacheByte:= cacheByte1);
	ELSE
		//second byte is within display
		cacheByte2 := GetCacheByte(address:= address + displayWidth);
		CASE mode OF
			LCD_MODES.CLEAR_BIT:
				cacheByte1 := cacheByte1 AND NOT MEM.LowByte(wValue:= tmpData);
				cacheByte2 := cacheByte2 AND NOT MEM.HighByte(wValue:= tmpData);
			LCD_MODES.SET_BIT:
				cacheByte1 := cacheByte1 AND NOT MEM.LowByte(wValue:= tmpMask);
				cacheByte2 := cacheByte2 AND NOT MEM.HighByte(wValue:= tmpMask);
				cacheByte1 := cacheByte1 OR MEM.LowByte(wValue:= tmpData);
				cacheByte2 := cacheByte2 OR MEM.HighByte(wValue:= tmpData);
			LCD_MODES.INVERT_BIT:
				cacheByte1 := cacheByte1 XOR MEM.LowByte(wValue:= tmpData);
				cacheByte2 := cacheByte2 XOR MEM.HighByte(wValue:= tmpData);
		END_CASE
		SetCacheByteRaw(address:= address, cacheByte:= cacheByte1);
		SetCacheByteRaw(address:= address + displayWidth, cacheByte:= cacheByte2);
	END_IF
END_IF
END_METHOD

METHOD SetSoftFont
VAR_INPUT
	font:SOFT_FONT_NUMS;
END_VAR
aktFont:=int_to_usint(limit(0,font,usint_to_int(SOFT_FONT_NUMS.last)-1) );//select form 0 to last
END_METHOD

METHOD WriteChar
VAR_INPUT
	c:USINT;
	mode: LCD_MODES;
END_VAR
VAR
	address:POINTER TO BYTE;
	i:USINT;
	mask:ARRAY[0..3] OF BYTE;
	unpackDWord:MEM.UnpackDWord;
	
END_VAR
address := softFontData[aktFont].data + (softFontData[aktFont].size * c); 

IF softFontData[aktFont].height <= 8 THEN
	unpackDWord(
	dwValue:= softFontData[aktFont].mask,
	byLLByte=> mask[0], 
	);
	//one byte font
	FOR i := 0 TO softFontData[aktFont].width - 1 DO
		SetByteCache(
			xpos:= cursorX + i, 
			ypos:= cursorY, 
			data:= address^, 
			mask := mask[0], 
			mode:= mode);
		address := address + 1;
	END_FOR
ELSIF softFontData[aktFont].height >8 AND softFontData[aktFont].height <= 16 THEN
	unpackDWord(
	dwValue:= softFontData[aktFont].mask,
	byLLByte=> mask[0],
	byLHByte=> mask[1] 
	);
	//two byte font
	FOR i := 0 TO softFontData[aktFont].width - 1 DO
		SetByteCache(
			xpos:= cursorX + i, 
			ypos:= cursorY, 
			data:= address^, 
			mask:= mask[0], 
			mode:= mode);
		address := address + 1;
		SetByteCache(
			xpos:= cursorX + i, 
			ypos:= cursorY + 8, 
			data:= address^, 
			mask:= mask[1], 
			mode:= mode);
		address := address + 1;
	END_FOR
ELSIF softFontData[aktFont].height >16 AND softFontData[aktFont].height <= 24 THEN
	unpackDWord(
	dwValue:= softFontData[aktFont].mask,
	byLLByte=> mask[0],
	byLHByte=> mask[1],
	byHLByte=> mask[2] 
	);
	//tree byte font
	FOR i := 0 TO softFontData[aktFont].width - 1 DO
		SetByteCache(
			xpos:= cursorX + i, 
			ypos:= cursorY, 
			data:= address^, 
			mask:= mask[0], 
			mode:= mode);
		address := address + 1;
		SetByteCache(
			xpos:= cursorX + i, 
			ypos:= cursorY + 8, 
			data:= address^, 
			mask:= mask[1], 
			mode:= mode);
		address := address + 1;
		SetByteCache(
			xpos:= cursorX + i, 
			ypos:= cursorY + 16, 
			data:= address^, 
			mask:= mask[2], 
			mode:= mode);
		address := address + 1;
	END_FOR
ELSIF softFontData[aktFont].height >24 THEN
	unpackDWord(
	dwValue:= softFontData[aktFont].mask,
	byLLByte=> mask[0],
	byLHByte=> mask[1],
	byHLByte=> mask[2],
	byHHByte=> mask[3] 
	);
	//four byte font
	FOR i := 0 TO softFontData[aktFont].width - 1 DO
		SetByteCache(
			xpos:= cursorX + i, 
			ypos:= cursorY, 
			data:= address^, 
			mask:= mask[0], 
			mode:= mode);
		address := address + 1;
		SetByteCache(
			xpos:= cursorX + i, 
			ypos:= cursorY + 8, 
			data:= address^, 
			mask:= mask[1], 
			mode:= mode);
		address := address + 1;
		SetByteCache(
			xpos:= cursorX + i, 
			ypos:= cursorY + 16, 
			data:= address^, 
			mask:= mask[2], 
			mode:= mode);
		address := address + 1;
		SetByteCache(
			xpos:= cursorX + i, 
			ypos:= cursorY + 24, 
			data:= address^, 
			mask:= mask[3], 
			mode:= mode);
		address := address + 1;

	END_FOR

END_IF

cursorX := cursorX + softFontData[aktFont].width;

//check for linefeed
IF cursorX + softFontData[aktFont].width > displayWidth THEN
	LineFeed();
END_IF
END_METHOD

METHOD FillBox
VAR_INPUT
	x1:USINT;
	y1:USINT;
	x2:USINT;
	y2:USINT;
	mode:LCD_MODES;
END_VAR
VAR
	i:USINT;
	temp:USINT;
	y:USINT;
END_VAR
IF x2 < x1 THEN
	//toggle x1 x2
	temp := x1;
	x1 := x2;
	x2 := temp;
END_IF

IF y2 < y1 THEN
	//toggle y1 y2
	temp := y1;
	y1 := y2;
	y2 := temp;
END_IF


//now draw box
FOR i := x1 TO x2  DO
	DrawLine(
	x1:= i, 
	y1:= y1, 
	x2:= i, 
	y2:= y2, 
	mode:= mode);
END_FOR
END_METHOD

METHOD LineFeed
VAR_INPUT
END_VAR
cursorX := cursorBaseX;
cursorY := cursorY + softFontData[aktFont].height;
END_METHOD

//Cursor mean upper left corner

METHOD SetCursor
VAR_INPUT
	x:USINT;
	y:USINT;
END_VAR
cursorX := x;
cursorBaseX := cursorX;

cursorY := y;
cursorBaseY := cursorY;
END_METHOD

END_FUNCTION_BLOCK

// Function Blocks/PCF8575OUT
FUNCTION_BLOCK PCF8575OUT EXTENDS I2C_BASE implements SetSlaveNum

VAR_INPUT
	outs: ARRAY[0..1] OF BYTE;
END_VAR
VAR
	lowOld:BYTE;
	hiOld:BYTE;
END_VAR

SUPER^();

METHOD Initialize : UDINT
VAR_INPUT
	wModuleType : UINT;
	dwInstance : UDINT;
	pConnector : POINTER TO IoConfigConnector;
END_VAR
VAR

END_VAR
SUPER^.Initialize(wModuleType, dwInstance, pConnector);


stateAfterError := RUN_DEVICE;
stateAfterInit := RUN_DEVICE;
END_METHOD

METHOD BeforeWriteOutputs : INT
VAR
	i: USINT;
	pyBuffer:ARRAY[0..2]OF BYTE;
END_VAR
SUPER^.BeforeWriteOutputs();

//GVL.callNum := 0;
IF checkInitMultiplex() THEN
	RETURN;
END_IF
CASE _iState OF


RUN_DEVICE:
	//requestWrite
	IF lowOld <> outs[0] OR hiOld <> outs[1] THEN
		writeRequest.request := TRUE;
	END_IF
	IF NOT checkWriteTimeMultiplex(ADR(writeRequest)) THEN
		RETURN;
	END_IF
	//reset request
	writeRequest.request := FALSE;
	//save old values
	lowOld := outs[0];
	hiOld := outs[1];
	checkWrite(ADR(outs),2);
	
END_CASE
END_METHOD


METHOD ResetWire
outs[0] := 255;
outs[1] := 255;
lowOld := outs[0];
hiOld := outs[1];
checkWrite(ADR(outs),2);
END_METHOD


METHOD SetSlaveEnableNum : SET_SLAVE_NUM_RETURN
VAR_INPUT
	num	: USINT;
END_VAR
IF _iState = RUN_DEVICE THEN
	IF num <8 THEN
		outs[0] := 255 AND NOT SHL(1, num);
	END_IF
	IF num >7 THEN
		outs[1] := 255 AND NOT SHL(1, num - 8);
	END_IF
	lowOld := outs[0];
	hiOld := outs[1];
	checkWrite(ADR(outs),2);
	IF _iState = RUN_DEVICE THEN
		SetSlaveEnableNum := SET_SLAVE_NUM_RETURN.NUM_IO;
	ELSE
		SetSlaveEnableNum := SET_SLAVE_NUM_RETURN.NUM_NIO;
	
	END_IF
END_IF
END_METHOD

END_FUNCTION_BLOCK

// Function Blocks/SI7021
FUNCTION_BLOCK SI7021 EXTENDS I2C_BASE
VAR_INPUT

END_VAR
VAR_OUTPUT
	myData:SI7021Data;
END_VAR
VAR


	controlRegister:BYTE;
	writeControlRegister:BOOL;
	operationMode:BYTE;
	//Time for next measurment
	NextMeasuerment: CAA.TICK;
	//time when i read next
	TimeToRead: CAA.TICK;
	//time to read in ms
	timePreset:UDINT;
	//time between measurments  in ms
	timeMeasurment:UDINT;
	//
	haveToRead: BOOL;
	//wait for done
	waitForDone: BOOL;
	//Time to read over
	TimeToReadOver: BOOL;
	//write request for command read humnity
	WriteRequestHuminity: BOOL;

	
	ReadHuminityErrorRate:DINT;
	ReadTempErrorRate:DINT;
	CRCErrorRate:DINT;
	WriteTime:CAA.TICK;
	ReadTime:CAA.TICK;
	WriteTempReadErrorRate:CAA.TICK;
	WriteHumninityReadErrorRate:CAA.TICK;
	crc:DWORD;
END_VAR
VAR_TEMP	
END_VAR

VAR CONSTANT 
	COMMAND_MEASURE_RH_HOLD_MASTER : BYTE := 16#E5;
	COMMAND_MEASURE_RH_NO_HOLD_MASTER : BYTE := 16#F5;
	COMMAND_MEASURE_TEMP_HOLD_MASTER : BYTE := 16#E3;
	COMMAND_MEASURE_TEMP_NO_HOLD_MASTER : BYTE := 16#F3;
	COMMAND_READ_TEMP_FROM_PREVIOUS_RH : BYTE := 16#E0;
	COMMAND_RESET : BYTE := 16#FE;
	COMMAND_WRITE_RESISTER_1 : BYTE := 16#E6;
	COMMAND_READ_RESISTER_1 : BYTE := 16#E7; 
	COMMAND_WRITE_HEATER_RESISTER : BYTE := 16#51;
	COMMAND_READ_HEATER_RESISTER : BYTE := 16#11;
	COMMAND_READ_ELECTRONIC_ID_1 : WORD := 16#FA0F;
	COMMAND_READ_ELECTRONIC_ID_2 : WORD := 16#FCC9;
	COMMAND_READ_FIRMWARE : WORD := 16#84B8; 
	

END_VAR

SUPER^();

CASE _iState OF
	RUN_DEVICE:;

END_CASE

METHOD AfterReadInputs : INT
VAR
	buffer:ARRAY[0..2] OF BYTE;
	buffercrc:ARRAY[0..3] OF BYTE;
	
END_VAR
SUPER^.AfterReadInputs();

